  bI_EnableBalance                          : ARRAY[1..iCIk_NB_INKBALANCE] OF BOOL;    (*enable balance*)
  sI_InkDensitySet                          : ARRAY[1..iCIk_NB_INKBALANCE] OF REAL;    (*Ink density TO convert [kg] TO [liter]*)
  sI_CorrectionValue                        : ARRAY[1..iCIk_NB_INKBALANCE] OF REAL;    (*Correction value for the MUX retrieved data*)
  sI_WarningLevelSet                        : ARRAY[1..iCIk_NB_INKBALANCE] OF REAL;    (*warning level on the balance in [liter]*)
  sI_ErrorlevelSet                          : ARRAY[1..iCIk_NB_INKBALANCE] OF REAL;    (*error level on the balance in [liter]*)

  lR_VarParamScannerId                      : ARRAY[1..iCIk_NB_INKBALANCE] OF UDINT;   (*varnish parameter scanner ID*)
  iR_VarParamIndex                          : ARRAY[1..iCIk_NB_INKBALANCE] OF UINT;    (*varnish parameter index*)
  bR_VarParamCompatibility                  : ARRAY[1..iCIk_NB_INKBALANCE, 1..10] OF BOOL; (*varnish parameter compatibility to other index*)
  fR_VarParamTemp                           : ARRAY[1..iCIk_NB_INKBALANCE] OF REAL;    (*varnish parameter temperature*)
  fR_VarParamMenc                           : ARRAY[1..iCIk_NB_INKBALANCE] OF REAL;    (*varnish parameter meniscus*)
  aR_VarParamWaveform                       : ARRAY[1..iCIk_NB_INKBALANCE] OF STRING;  (*varnish parameter waveform*)
  iR_VarParamTimer                          : ARRAY[1..iCIk_NB_INKBALANCE] OF UINT;    (*varnish parameter timer*)
  fR_VarParamDensity                        : ARRAY[1..iCIk_NB_INKBALANCE] OF REAL;    (*varnish parameter density*)
  fR_VarParamViscosity                      : ARRAY[1..iCIk_NB_INKBALANCE] OF REAL;    (*varnish parameter viscosity*)
  iR_VarParamColorId                        : ARRAY[1..iCIk_NB_INKBALANCE] OF UINT;    (*varnish parameter color ID*)

  aI_CalibrateFrameText1                    : ARRAY[1..iCIk_NB_INKBALANCE] OF STRING;  (*Calibration string variable for text 1*)
  aI_CalibrateFrameText2                    : ARRAY[1..iCIk_NB_INKBALANCE] OF STRING;  (*Calibration string variable for text 2*)

  fR_BalanceOffset                          : ARRAY[1..iCIk_NB_INKBALANCE] OF REAL;   (*Calibration value for empty tank*)


(*Last entry----retain (remanent) variables of PRG_INK and realated modules*)
  aL_Pattern                                : UDINT;  (*check pattern for rem validity*)
END_STRUCT
END_TYPE

// ---- DUTs/Projects/Structures/ST_REM_VAR_M.TcDUT
TYPE ST_REM_VAR_M :
(*************************************************************************************************)
(*  FILENAME:    ST_REM_VAR_M.EXP                                                                *)
(*  PROJECT:     CALMAR PUPLC                                                                    *)
(*  COPYRIGHT:   All rights reserved (c) Wifag//Polytype, Fribourg/Switzerland (2016)            *)
(*  ENVIRONMENT: TwinCAT PLC                                                                     *)
(*  VERSION:     <version>                                                                       *)
(*************************************************************************************************)
(*  DESCRIPTION:                                                                   <description> *)
(*    Structure of remanent variables.                                                           *)
(*                                                                                </description> *)
(*************************************************************************************************)

STRUCT
  (*Clean Head*)
  (*************************************************************************************************)
  fRCH_Position_A                           : REAL;
  fRCH_Position_B                           : REAL;
  fRCH_Position_p1                          : REAL;
  fRCH_Position_p2                          : REAL;
  fRCH_PlaceSpeed                           : REAL;
  fRCH_WorkSpeed                            : REAL;
  fRCH_ServiceSpeed                         : REAL;

  lRCH_OffsetEncoder                        : DINT;
  

  lR_ToleranceLenPx                         : DINT;

(*Last entry----retain (remanent) variables of PRG_MACHINE and realated modules*)
  aL_Pattern                                : UDINT;  (*check pattern for rem validity*)
END_STRUCT
END_TYPE

// ---- DUTs/Projects/Structures/ST_REM_VAR_P.TcDUT
TYPE ST_REM_VAR_P :
(*************************************************************************************************)
(*  FILENAME:    ST_REM_VAR_P.EXP                                                                *)
(*  PROJECT:     CALMAR PUPLC                                                                    *)
(*  COPYRIGHT:   All rights reserved (c) Wifag//Polytype, Fribourg/Switzerland (2016)            *)
(*  ENVIRONMENT: TwinCAT PLC                                                                     *)
(*  VERSION:     <version>                                                                       *)
(*************************************************************************************************)
(*  DESCRIPTION:                                                                   <description> *)
(*    Structure of remanent variables.                                                           *)
(*                                                                                </description> *)
(*************************************************************************************************)

STRUCT
  (*PU*)
  //iL_ResolutionPhPx                      : ARRAY [1..iCPr_NB_PU] OF INT;    (*printhead pixel resolution [dpi]*)
  //fL_ResolutionEncoder                   : ARRAY [1..iCPr_NB_PU] OF LREAL;  (*resolution of encoder [um/increment]*)
  //iL_ResolutionSubPx                     : ARRAY [1..iCPr_NB_PU] OF INT;    (*subpixel pulse resolution [pulse/px]*)
  //fL_Pg_xOffset                          : ARRAY [1..iCPr_NB_PG] OF LREAL;  (*static offset of print group from start detection [m]*)
  //fL_Pg_vStartShiftFactor                : ARRAY [1..iCPr_NB_PU] OF LREAL;  (*shift of virtual start signal value from detection towards print group [m]*)
  //fL_Pg_vStartShiftOffset                : ARRAY [1..iCPr_NB_PU] OF LREAL;  (*shift of virtual start signal value from detection towards print group [m]*)
  //fL_SubstrateLen                        : ARRAY [1..iCPr_NB_PU] OF REAL;   (*length of substrate [m]*)

  bL_sAdsPrintUnit_bI_Enable             : ARRAY [1..iCPr_NB_PU] OF BOOL;
  lL_sAdsPrintUnit_sI_ShiftJobX          : ARRAY [1..iCPr_NB_PU] OF DINT;   (*Job(Unit) shift X in Pixel*)
  lL_sAdsPrintUnit_sI_ShiftJobY          : ARRAY [1..iCPr_NB_PU] OF DINT;   (*Job(Unit) shift Y in Pixel*)

  (*PM*)
  //fL_ResolutionEncoderPM                 : ARRAY [1..iCPr_NB_PM] OF LREAL;  (*resolution of encoder [um/increment]*)

  (*PG*)
  rL_sAdsPrintGroup_bI_Enable            : ARRAY [1..iCPr_NB_PG] OF BOOL;
  rL_sAdsPrintGroup_iO_PositionX         : ARRAY [1..iCPr_NB_PG] OF DINT;
  rL_sAdsPrintGroup_iO_StartPositionX    : ARRAY [1..iCPr_NB_PG] OF DINT;

  (*PC*)
  rL_sAdsPrintController                 : ARRAY [1..iCPr_NB_PC] OF BOOL;
  rL_sAdsPrintControllerHeater           : ARRAY [1..iCPr_NB_PC] OF BOOL;   (*Enable heater*)
  rL_sAdsPrintControllerPrint            : ARRAY [1..iCPr_NB_PC] OF BOOL;   (*Enable print*)

  (*PH*)
  rL_sAdsPrintHead_bI_Enable             : ARRAY [1..iCPr_NB_PH] OF BOOL;
  rL_sAdsPrintHead_iO_PositionX          : ARRAY [1..iCPr_NB_PH] OF DINT;
  rL_sAdsPrintHead_iO_StartPositionX     : ARRAY [1..iCPr_NB_PH] OF DINT;
  rL_sAdsPrintHead_iO_StartPositionY     : ARRAY [1..iCPr_NB_PH] OF DINT;
  rL_sAdsPrintHead_aI_MaskFileName       : ARRAY [1..iCPr_NB_PH] OF STRING; (*File name of sticking mask file*)
  rL_sAdsPrintHead_aI_WaveFileName       : ARRAY [1..iCPr_NB_PH] OF STRING; (*File name of waveform configuration file*)
  rL_sAdsPrintHead_fI_VoltScale          : ARRAY [1..iCPr_NB_PH] OF REAL;   (*File name of waveform configuration file*)
  
  bL_WithMark                            : BOOL;  (*use mark detection*)
  fL_MarkLength                          : REAL;  (*mark length*)
  fL_MarkHeigth                          : REAL;  (*mark width*)
  //fL_HeadGap                             : REAL;

  //bL_SpeedCompensationEnable             : BOOL;
  //fL_SpeedCompensationFactor             : REAL;
  //fL_SpeedCompensationBase               : REAL;

  fR_DriftTimeShift                      : LREAL;
  
  //iL_MonitorTempPH                       : INT;  (*Monitor level of temperature*)

(*Last entry----retain (remanent) variables of PRG_PRINT and realated modules*)
  aL_Pattern                             : UDINT;  (*check pattern for rem validity*)
END_STRUCT
END_TYPE

// ---- POUs/Products/Print_Weu/E_PosDomain.TcTLEO
{attribute 'qualified_only'}
{attribute 'strict'}
TYPE E_PosDomain :
(
	default := 0,
  master_pos := 1,
//  cycle_pos := 2
  pos_px      := 2     // position in [px]
) UINT;
END_TYPE

// ---- POUs/Products/Print_Weu/Mark/ST_MarkDefinition.TcDUT
TYPE ST_MarkDefinition :
STRUCT
  nId : DINT;             // mark id (array index)
  fHeight : LREAL;        // [m] mark height (size Y)
  fTrLength : LREAL;      // [m] triangle lenght
  fSqLength : LREAL;      // [m] square length ( square + triangle lengh = sizeX)
  fPosX : LREAL;          // [m] position X offset from 0/0
  fPosY : LREAL;          // [m] position Y offset from 0/0
  bInvertedX : BOOL;      // flipped in X axis (prior bMarksInverted)
  //bInvertedY : BOOL;      // flipped in Y axis
  //state
  sState : ST_MarkState;  // mark detection state
  //view
  bShow : BOOL;
  nMove : DINT;
END_STRUCT 
END_TYPE

// ---- POUs/Products/Print_Weu/Mark/ST_MarkState.TcDUT
TYPE ST_MarkState :
STRUCT
  bSet        : BOOL;     // mark was set & valid (detected)
  bMissed     : BOOL;     // mark was missing (+internally generated)
  bInArea     : BOOL;     // mark withing ok area
  dx          : LREAL;    // x displacement [m]
  dy          : LREAL;    // y displacement [m]
  fLengthReal : LREAL;    // real detected mark length [m]
  nPosXReal   : DINT;     // detected position X absolute [SubPx]
END_STRUCT
END_TYPE

// ---- POUs/Products/Print_Weu/ST_MappingDefinition.TcDUT
(*
  Hardware mapping definition.
*)
TYPE ST_MappingDefinition :
STRUCT
  // absolute hw mapping
  nPhInst : UDINT := 1;      // ph hw instance selection
  nPcInst : UDINT := 1;      // pc hw instance selection
  // module internal mapping (relative to given nPm)
  nPm     : UDINT := 1;      // to pm x
  nPg     : UDINT := 1;      // to pg in pm x
  nPa     : UDINT := 1;      // to pa in pg
  nPs     : UDINT := 1;      // to ps in pa
  nPc     : UDINT := 1;      // to pc in pm
  nPcCh   : UDINT := 1;      // to pc channel of pc 1-4
END_STRUCT
END_TYPE

// ---- POUs/Products/Print_Weu/ST_ModuleMachineInterface_IN.TcDUT
TYPE ST_ModuleMachineInterface_IN :
STRUCT
  // Inputs (from machine)
  bEStop                  : BOOL;             // EStop active
  bSleep                  : BOOL;             // Sleep active
  bSafetyCoverOk          : BOOL;             // Safety cover OK
  bServiceDoorsOk         : BOOL;             // Safety Doors OK
  bExhaustVacuumWarning   : BOOL;             // Vacuum warning level reached
  bExhaustVacuumError     : BOOL;             // Vacuum error level reached
  bExhaustFUError         : BOOL;             // ??? (obsolete?)
  bDriftControlError      : BOOL;             // (obsolete) remove?
  bDriftControlMissMarks  : BOOL;             // (obsolete) remove?
  bSafetyOk               : BOOL;              // generic safty ok
  
  // new
  bUnitInPrintPosition    : BOOL;             // Print module in print position
  bEngaged                : BOOL;             // Print module engaged
  bPrintEnabled           : BOOL;             // Printing enabled
  
  // other
  fSubstrateThickness     : LREAL := 0.000_1; // Substrate thickness [m]
  fSubstrateLen           : LREAL;            // Substrate length [m]
  fWebStretchCalculated   : LREAL;            // Web strech factor converted
  fLateralRegister        : LREAL;            // Lateral regster [m]
  fModule2ToModule3       : LREAL;            // Distance between Module 2 and 3 [m]
  bTargetSpeedReached     : BOOL;             // Target speed reached
  fNeutralFibreFactor     : LREAL;            // Neutral fibre factor [%]

END_STRUCT
END_TYPE

// ---- POUs/Products/Print_Weu/ST_ModuleMachineInterface_OUT.TcDUT
TYPE ST_ModuleMachineInterface_OUT :
STRUCT
  // Outputs (to Machine)
  fSpeed                : LREAL;            // Current module speed [m/s]
  bMoving               : BOOL;             // substrate/module is moving
  nPrintMarkPosBits     : WORD;             // Print mark position (bit coded)
  fMaxSpeed             : LREAL;            // Max. possible print module speed [m/s]
  bSpeedExeeded         : BOOL;             // Module speed exeeded;
END_STRUCT
END_TYPE

// ---- VISUs/Projects/Print/ST_ButtonFrameSel_Def.TcDUT
TYPE ST_ButtonFrameSel_Def :
STRUCT
  sImgId       : STRING;           // image id (to show)
  nFrameIdx    : UINT;             // frame index [0..x], index to select on click
  pFrameSelect : POINTER TO UINT;  // pointer to frame selection variable (variable to write to change the selected frame)
  sVisuName    : T_MaxString;      // visualisation name
END_STRUCT
END_TYPE

// ---- GVLs/Configuration/CONFIGURATION.TcGVL
{attribute 'Tc2GvlVarNames'}
VAR_GLOBAL CONSTANT
(*************************************************************************************************)
(*  FILENAME:    CONFIGURATION.EXP                                                               *)
(*  PROJECT:     CALMAR PUPLC                                                                    *)
(*  COPYRIGHT:   All rights reserved (c) Wifag//Polytype, Fribourg/Switzerland (2016)            *)
(*  ENVIRONMENT: TwinCAT PLC                                                                     *)
(*  VERSION:     <version>                                                                       *)
(*************************************************************************************************)
(*  DESCRIPTION:                                                                   <description> *)
(*    Configuration data system.                                                                 *)
(*                                                                                </description> *)
(*************************************************************************************************)

(*************************************************************************************************)
(*Configuration System*)
(*************************************************************************************************)
  iCSYS_GEN_BLOCK_MAP_CONFIG        : UINT := 0;   (*Configuration FB_GEN_BLOCK_MAPPING*)
                                                   (*Bit0: use extended block id then UINT :=  1; (iC_CFG_BIT_EXT_ID) *)


(*************************************************************************************************)
(*Configuration InkSystem*)
(*************************************************************************************************)

(*ADS*)
(*************************************************************************************************)
  iCIk_NB_BLOCK_TYPES               : INT := 10;   (*Number of different ADS block types*)


(*GENERAL*)
(*************************************************************************************************)
  (*Number of print station*)
  iCIk_NB_PRINT_STA                 : INT := 1;    (*Number of print station*)


(*DEGASSING*)
(*************************************************************************************************)
  iCIk_NB_DGAS                      : INT := 1;    (*Number of dgas controller*)

  bCIk_INK_DEGASSING_EXISTING       : BOOL := TRUE;  (*Degassing of ink existing*)


(*MENISCUS*)
(*************************************************************************************************)
  (*Number of menc controller*)
  iCIk_NB_MENC                      : INT := 1;    (*Number of menc controller*)

  (*Mapping main meniscus*)
  iCIk_MAP_MAIN_MENC_PURGE          : ARRAY [1..iCIk_NB_MENC] OF INT := [1];  (*Mapping main menc to purge controller*)

  (*Number of sub menc controller*)
  iCIk_NB_SUB_MENC                  : INT := 2;    (*Number of sub menc controller*)

  (*Number of menc controller per station*)
  iCIk_NB_MENC_STA                  : INT := 3;    (*Number of menc controller per station (iCIk_NB_MENC + iCIk_NB_SUB_MENC)*)

  (*Mapping sub meniscus*)
  iCIk_MAP_SUB_MENC_MAIN_MENC       : ARRAY [1..iCIk_NB_SUB_MENC] OF INT := [1,1];  (*Mapping sub menc to main menc*)
  iCIk_MAP_SUB_MENC_PURGE           : ARRAY [1..iCIk_NB_SUB_MENC] OF INT := [1,2];  (*Mapping sub menc to purge controller*)
  iCIk_MAP_SUB_MENC_HTG             : ARRAY [1..iCIk_NB_SUB_MENC] OF INT := [1,2];  (*Mapping sub menc to headertank group*)


(*PURGE - GLOBAL*)
(*************************************************************************************************)
  iCIk_NB_PURGE_CONTR               : INT := 2;    (*Number of purge controller*)
  iCIk_NB_PURGE_GROUP               : INT := 4;    (*Number of purge groups*)

  (*Purge controller existing*)
  bCIk_PURGE_CONTR_EXIST            : ARRAY [1..iCIk_NB_PURGE_CONTR] OF BOOL := [TRUE,TRUE];

  (*Purge group existing*)
  bCIk_PURGE_GROUP_EXIST            : ARRAY [1..iCIk_NB_PURGE_GROUP] OF BOOL := [TRUE,TRUE,TRUE,TRUE];

  (*Mapping purge group*)
  cCIk_MAP_PURGE_GROUP_CONTR        : ARRAY [1..iCIk_NB_PURGE_GROUP] OF BYTE := [1,1,2,2];  (*Mapping purge group to purge controller*)
  cCIk_MAP_PURGE_GROUP_PURGE_STA    : ARRAY [1..iCIk_NB_PURGE_GROUP] OF BYTE := [1,2,1,2];  (*Mapping purge group to purge station*)

  (*Purge for White is working with a special sequence*)
  bCIk_PURGE_CONTR_SEQUENCE         : ARRAY [1..iCIk_NB_PURGE_CONTR] OF BOOL := [FALSE,FALSE];
  bCIk_MAP_PURGE_CONTR_SEQ_MENC_NEG : ARRAY [1..iCIk_NB_PURGE_CONTR] OF BYTE := [2,2];
  bCIk_MAP_PURGE_CONTR_SEQ_MENC_POS : ARRAY [1..iCIk_NB_PURGE_CONTR] OF BYTE := [3,3];

  bCIk_PURGE_SEQUENCE_MAIN_VALVE    : BOOL := TRUE;   (*Use main or sub valve for sequence*)
  bCIk_PURGE_CONTROLLER_SEQUENTIAL  : BOOL := FALSE;  (*Purge controller process sequential*)
  bCIk_PURGE_CYCLE_CLOSE_PH_VALVE   : BOOL := FALSE;  (*Close valve PHin and PHout between the cycles*)
  bCIk_PURGE_PRESSURE_LINE          : BOOL := TRUE;   (*Purge pressure is connected direct to a pressure line*)


(*INK*)
(*************************************************************************************************)
  iCIk_NB_HEADERTANK                : INT := 4;       (*Number of headertanks*)
  iCIk_NB_HEADERTANK_GROUP          : INT := 2;       (*Number of headertank groups*)

  (*Headertank existing*)
  (*'White Recirculation','White front','White back','Cyan','Magenta','Yellow','Black'*)
  bCIk_HEADERTANK_EXIST             : ARRAY [1..iCIk_NB_HEADERTANK] OF BOOL := [ TRUE, TRUE, TRUE, TRUE];
  bCIk_HEADERTANK_FILL_CLEANER      : ARRAY [1..iCIk_NB_HEADERTANK] OF BOOL := [FALSE,FALSE,FALSE,FALSE];
  bCIk_HEADERTANK_REFUSE            : ARRAY [1..iCIk_NB_HEADERTANK] OF BOOL := [FALSE,FALSE,FALSE,FALSE];
  bCIk_HEADERTANK_CHANGE            : ARRAY [1..iCIk_NB_HEADERTANK] OF BOOL := [ TRUE, TRUE, TRUE, TRUE];
  bCIk_HEADERTANK_FILL              : ARRAY [1..iCIk_NB_HEADERTANK] OF BOOL := [ TRUE, TRUE, TRUE, TRUE];
  bCIk_HEADERTANK_FLUSH             : ARRAY [1..iCIk_NB_HEADERTANK] OF BOOL := [ TRUE, TRUE, TRUE, TRUE];

  (*Mapping headertank*)
  iCIk_MAP_HEADERTANK_DGAS          : ARRAY [1..iCIk_NB_HEADERTANK] OF INT := [1,1,1,1];  (*Mapping headertank to degass*)
  iCIk_MAP_HEADERTANK_MENC_STA      : ARRAY [1..iCIk_NB_HEADERTANK] OF INT := [2,2,3,3];  (*Mapping headertank to menc station*)
  iCIk_MAP_HEADERTANK_INK           : ARRAY [1..iCIk_NB_HEADERTANK] OF INT := [1,1,2,2];  (*Mapping headertank to ink*)
  iCIk_MAP_HEADERTANK_INK_LEVEL     : ARRAY [1..iCIk_NB_HEADERTANK] OF INT := [1,2,3,4];  (*Mapping headertank to ink level sensor*)
  iCIk_MAP_HEADERTANK_INK_PUMP      : ARRAY [1..iCIk_NB_HEADERTANK] OF INT := [1,2,3,4];  (*Mapping headertank to ink pump*)
  iCIk_MAP_HEADERTANK_PURGE_CONTR   : ARRAY [1..iCIk_NB_HEADERTANK] OF INT := [1,1,2,2];  (*Mapping headertank to purge controller*)
  iCIk_MAP_HEADERTANK_PURGE_GROUP   : ARRAY [1..iCIk_NB_HEADERTANK] OF INT := [1,2,3,4];  (*Mapping headertank to purge group*)
  iCIk_MAP_HEADERTANK_PURGE_GROUPIDX: ARRAY [1..iCIk_NB_HEADERTANK] OF INT := [1,2,1,2];  (*Mapping headertank to purge group*)
  iCIk_MAP_HEADERTANK_STORAGE_PUMP  : ARRAY [1..iCIk_NB_HEADERTANK] OF INT := [1,2,3,4];  (*Mapping headertank to storagetank pump*)
  iCIk_MAP_HEADERTANK_CLEANER_PUMP  : ARRAY [1..iCIk_NB_HEADERTANK] OF INT := [1,1,2,2];  (*Mapping headertank to cleaner pump*)
  iCIk_MAP_HEADERTANK_RETURN_FLOW   : ARRAY [1..iCIk_NB_HEADERTANK] OF INT := [1,1,2,2];  (*Mapping headertank to return flow*)
  iCIk_MAP_HEADERTANK_TEMP_CONTR    : ARRAY [1..iCIk_NB_HEADERTANK] OF INT := [1,2,3,4];  (*Mapping headertank to Temp controller*)
  iCIk_MAP_HEADERTANK_HT_GROUP      : ARRAY [1..iCIk_NB_HEADERTANK] OF INT := [1,1,2,2];  (*Mapping headertank to headertank group*)

  (*Storagetank*)
  iCIk_NB_INK                       : INT  := 2;    (*Number of ink*)
  iCIk_NB_INKSTORAGE_TANK           : INT  := 3;    (*Number of storage tanks incl conservation tank*)
  iCIk_NB_INKSTORAGE_TANK_MAX       : INT  := CalmarCompInkSystem.GVL_InkDef.iCIk_NB_INKSTORAGE_TANK_MAX;    (*Max number of storage tanks*)
  iCIk_NB_INKSTORAGE_TANK_MIXER     : INT  := 2;    (*Number of storage tank mixer (not existing here)*)
  iCIk_NB_INKSTORAGE_TANK_PUMP      : INT  := 4;    (*e.g. iCIk_NB_HEADERTANK*)
  iCIk_STORAGE_TANK_PUMP_SETPOINT   : BOOL := FALSE; (*Pump speed controlled by a set point or fix*)
  iCIk_MAP_STORAGE_TANK_BALANCE     : ARRAY [1..iCIk_NB_INK] OF INT := [1,2];  (*Mapping storage tank to balances*)

  (*Ink storage tank existing, order see aC_STORAGETANK_NAME_DETAIL*)
  bCIk_INKSTORAGE_TANK_EXIST        : ARRAY [1..iCIk_NB_INKSTORAGE_TANK] OF BOOL := [TRUE,TRUE,TRUE];
  bCIk_INKSTORAGE_MIXER_EXIST       : ARRAY [1..iCIk_NB_INKSTORAGE_TANK] OF BOOL := [FALSE,FALSE,FALSE];
  iCIk_MAP_INKSTORAGE_MIXER         : ARRAY [1..iCIk_NB_INKSTORAGE_TANK] OF INT  := [    1,    2,    3];
  bCIk_MIXER_FEEDBACK_EXIST         : BOOL := FALSE;


  (*Number of ink pumps*)
  iCIk_NB_INK_PUMPS                 : INT := 10;  (*Number of ink pumps in total*)

  iCIk_NB_CLEANER_PUMPS             : INT := 2;   (*Number of cleaner pumps*)
  iCIk_CLEANER_PUMP_SETPOINT        : ARRAY [1..iCIk_NB_CLEANER_PUMPS]     OF BOOL := [FALSE,FALSE];  (*Pump speed controlled by a set point or fix*)

  iCIk_NB_RETURN_FLOW_UNITS         : INT  := 2;      (*Number of retrun flow units*)
  iCIk_RETURN_FLOW_PUMP_SETPOINT    : BOOL := FALSE;  (*Pump speed controlled by a set point or fix*)

  (*Number of ink level sensor*)
  iCIk_NB_INK_LEVEL_SENSOR          : INT := 6;   (*Number of ink level sensor*)
	iCIk_NB_INK_LEVEL_SENSOR_CIRCL    : INT := 1;   (*Number of ink level sensor for circulation*)


(*TEMP*)
(*************************************************************************************************)
  (*Number of heating*)
  iCIk_NB_TEMP_CONTR                : INT := 8;   (*Sum number of heating controllers*)
  iCIk_NB_TEMP_HYS                  : INT := 8;   (*Number of heating controller with hysteris*)

  (*Mapping temp*)
  iCIk_MAP_TEMP_INK                 : ARRAY [1..iCIk_NB_TEMP_CONTR] OF INT := [1,1,2,2,1,1,2,2];  (*Mapping temp to ink*)
  iCIk_MAP_TEMP_HT                  : ARRAY [1..iCIk_NB_TEMP_CONTR] OF INT := [1,2,3,4,1,2,3,4];  (*Mapping temp to ink*)
  iCIk_MAP_TEMP_PG                  : ARRAY [1..iCIk_NB_TEMP_CONTR] OF INT := [1,2,3,4,1,2,3,4];  (*Mapping temp to print group*)

  
(*BALANCE*)
(*************************************************************************************************)
  bCIk_BALANCE_EXISTING             : BOOL := TRUE;  (*Balance system existing*)

  cCIk_NB_BALANCE_CHANNELS          : BYTE:= 8;   (*Number of balance channels per MUX*)
  iCIk_NB_INKBALANCE                : INT := 2;   (*Number of used balance channels*)
  iCIk_NB_BALANCE_MUX               : INT := 1;   (*Number of balance MUX*)

  cCIk_BALANCE_MUX_ID               : ARRAY [1..iCIk_NB_BALANCE_MUX, 0..2] OF BYTE := [48,48,49]; (*Balance ASCII MUX ID 001*)

  (*Balance channel existing*)
  bCIk_INKBALANCE_EXIST             : ARRAY [1..iCIk_NB_INKBALANCE] OF BOOL := [TRUE, TRUE];

  (*Mapping balance*)
  cCIk_MAP_BALANCE_BALANCE_MUX      : ARRAY [1..iCIk_NB_INKBALANCE] OF BYTE := [1,1];        (*Mapping balance/storage tank to balance MUX*)
  cCIk_MAP_BALANCE_BALANCE_CHANNEL  : ARRAY [1..iCIk_NB_INKBALANCE] OF BYTE := [0,1];        (*Mapping balance/storage tank to balance channel*)

  iCIk_NB_COUNT_SEND_WARNING        : INT := 3;       (*Count of 'send data error' messages till warning*)
  iCIk_NB_COUNT_MOTION_WARNING      : INT := 10000;   (*Count of 'in motion' messages till warning*)
  iCIk_NB_COUNT_NC_WARNING          : INT := 5;       (*Count of 'not connected' messages till warning*)

  (*Messages*)
  iCIk_NB_BALANCE_MSG               : INT := 15;      (*Number of messages per balance*)


//BALANCE wiedre altes System!
  (*If no balance system existing iCIk_NB_INKBALANCE should nevertheless set to >0*)
	(*Number of balance (at least 1 for dummy)*)
  iCIk_BALANCE_POWER_SUPPLY         : INT  := 5;     (*Power supply of balances [V]*)
	fCIk_BALANCE_RATED_OUTPUT         : REAL := 3.0;   (*[mV/V]*)
	fCIk_BALANCE_RATED_CAPACITY       : REAL := 10.0;  (*[kg]*)
	fCIk_BALANCE_REFUSE_FULL          : REAL := 9.0;   (*[kg]*)
	fCIk_BALANCE_CLEANER_EMPTY        : REAL := 1.0;  (*[kg]*)

  
(*************************************************************************************************)
(*Configuration Machine                                                                          *)
(*************************************************************************************************)

(*ADS*)
(*************************************************************************************************)
  iCMa_NB_BLOCK_TYPES               : INT := 3;    (*Number of different ADS block types*)


(*GENERAL*)
(*************************************************************************************************)
  (*DEVICE COUNT*)
  iCMa_NB_Ax                        : INT := 3;      (*Number of axes*)
  iCMa_NB_Cp                        : INT := 2;      (*Number of cleaning process controllers*)
  iCMa_NB_Ca                        : INT := 8;      (*Number of clean axes: 4 per module*)
  iCMa_NB_Ma                        : INT := 1;      (*Number of machines*)

  (*Mapping GROUP*)
  iCPr_MAP_Cp_CuAxis                : ARRAY [1..iCMa_NB_Cp] OF INT := [1,5];    (*Mapping cleaning process to CU axis ADS*)
  iCPr_MAP_Cp_ChAxis                : ARRAY [1..iCMa_NB_Cp] OF INT := [2,6];    (*Mapping cleaning process to CH axis ADS*)
  iCPr_MAP_Cp_PuAxis                : ARRAY [1..iCMa_NB_Cp] OF INT := [3,7];    (*Mapping cleaning process to PU axis ADS*)
  iCPr_MAP_Cp_InkInterface          : ARRAY [1..iCMa_NB_Cp] OF INT := [4,8];    (*Mapping cleaning process to ink interface ADS*)

  (*Messages*)
  iCMa_NB_MSG                       : INT := 31;    (*Number of messages per machine*)

END_VAR

// ---- GVLs/Configuration/Configuration_Print.TcGVL
//{attribute 'qualified_only'}
{attribute 'Tc2GvlVarNames'}
VAR_GLOBAL CONSTANT
(*************************************************************************************************)
(*Configuration Print*)
(*************************************************************************************************)

(*ADS*)
(*************************************************************************************************)
iCPr_NB_BLOCK_TYPES               : INT := 6;    (*Number of different ADS block types*)

(*Print*)
nC_PrintResolution                : UDINT := 600;     (*Print resolutions native*)
nC_SubPixelResolution             : UDINT := 32;      (*SubPixel resolution, resolution extension of print resolution*)
nC_MemorySectionWidth             : UDINT := 16#800;  (*NIOS Memory section width/height*)
nC_MemorySectionDepth             : UDINT := 16#6000; (*NIOS Memory section depth/length*)
nC_YShiftOffset                   : UDINT := (nC_MemorySectionWidth - GVL_PrintDef.RIGEN5.iC_Ph_Width) / 2;  // [px] 384px for RICOH_GEN5



(*DEVICE COUNT*)
iCPr_NB_PH                        : INT := 24;  (*Number of printheads*)
iCPr_NB_PC                        : INT := 8;   (*Number of printhead controllers*)
iCPr_NB_PG                        : INT := 4;   (*Number of printhead groups*)
iCPr_NB_PM                        : INT := 2;   (*Number of print modules*)
iCPr_NB_PU                        : INT := 1;   (*Number of print units*)
iCPr_NB_SUBSTRATE_DEVICES         : INT := 1;   (*Number of substrate control devices*)
iCPr_NB_ASPECT                    : INT := 1;   (*Number of aspect definitions*)

iCPr_PH_MAPPING                   : ARRAY[1..iCPr_NB_PH] OF ST_MappingDefinition := 
[ 
  // PM 1 - NOTE: nPC global, nPcPc per pc, other values relative to PM
  (nPhInst := 1,  nPcInst := 1, nPm := 1, nPg := 1, nPa := 1, nPs := 1, nPc := 1, nPcCh := 1),    // 1
  (nPhInst := 2,  nPcInst := 1, nPm := 1, nPg := 1, nPa := 1, nPs := 1, nPc := 1, nPcCh := 2),    // 2
  (nPhInst := 3,  nPcInst := 1, nPm := 1, nPg := 1, nPa := 1, nPs := 1, nPc := 1, nPcCh := 3),    // 3
  (nPhInst := 4,  nPcInst := 2, nPm := 1, nPg := 1, nPa := 1, nPs := 1, nPc := 2, nPcCh := 1),    // 4
  (nPhInst := 5,  nPcInst := 2, nPm := 1, nPg := 1, nPa := 1, nPs := 1, nPc := 2, nPcCh := 2),    // 5
  (nPhInst := 6,  nPcInst := 2, nPm := 1, nPg := 1, nPa := 1, nPs := 1, nPc := 2, nPcCh := 3),    // 6
  (nPhInst := 7,  nPcInst := 3, nPm := 1, nPg := 2, nPa := 1, nPs := 1, nPc := 3, nPcCh := 1),    // 7
  (nPhInst := 8,  nPcInst := 3, nPm := 1, nPg := 2, nPa := 1, nPs := 1, nPc := 3, nPcCh := 2),    // 8
  (nPhInst := 9,  nPcInst := 3, nPm := 1, nPg := 2, nPa := 1, nPs := 1, nPc := 3, nPcCh := 3),    // 9
  (nPhInst := 10, nPcInst := 4, nPm := 1, nPg := 2, nPa := 1, nPs := 1, nPc := 4, nPcCh := 1),    // 10
  (nPhInst := 11, nPcInst := 4, nPm := 1, nPg := 2, nPa := 1, nPs := 1, nPc := 4, nPcCh := 2),    // 11
  (nPhInst := 12, nPcInst := 4, nPm := 1, nPg := 2, nPa := 1, nPs := 1, nPc := 4, nPcCh := 3),    // 12
  // PM 2 - NOTE: nPC global, nPcPc per pc, other values relative to PM
  (nPhInst := 13, nPcInst := 5, nPm := 2, nPg := 1, nPa := 1, nPs := 1, nPc := 1, nPcCh := 1),    // 13
  (nPhInst := 14, nPcInst := 5, nPm := 2, nPg := 1, nPa := 1, nPs := 1, nPc := 1, nPcCh := 2),    // 14
  (nPhInst := 15, nPcInst := 5, nPm := 2, nPg := 1, nPa := 1, nPs := 1, nPc := 1, nPcCh := 3),    // 15
  (nPhInst := 16, nPcInst := 6, nPm := 2, nPg := 1, nPa := 1, nPs := 1, nPc := 2, nPcCh := 1),    // 16
  (nPhInst := 17, nPcInst := 6, nPm := 2, nPg := 1, nPa := 1, nPs := 1, nPc := 2, nPcCh := 2),    // 17
  (nPhInst := 18, nPcInst := 6, nPm := 2, nPg := 1, nPa := 1, nPs := 1, nPc := 2, nPcCh := 3),    // 18
  (nPhInst := 19, nPcInst := 7, nPm := 2, nPg := 2, nPa := 1, nPs := 1, nPc := 3, nPcCh := 1),    // 19
  (nPhInst := 20, nPcInst := 7, nPm := 2, nPg := 2, nPa := 1, nPs := 1, nPc := 3, nPcCh := 2),    // 20
  (nPhInst := 21, nPcInst := 7, nPm := 2, nPg := 2, nPa := 1, nPs := 1, nPc := 3, nPcCh := 3),    // 21
  (nPhInst := 22, nPcInst := 8, nPm := 2, nPg := 2, nPa := 1, nPs := 1, nPc := 4, nPcCh := 1),    // 22
  (nPhInst := 23, nPcInst := 8, nPm := 2, nPg := 2, nPa := 1, nPs := 1, nPc := 4, nPcCh := 2),    // 23
  (nPhInst := 24, nPcInst := 8, nPm := 2, nPg := 2, nPa := 1, nPs := 1, nPc := 4, nPcCh := 3)     // 24
];


(*UNIT*)
iCPr_NB_PG_UNIT                   : INT := 4;   (*Number of groups in unit1*)

(*Mapping MODULE*)
iCPr_MAP_PM_PG                    : ARRAY [1..iCPr_NB_PM] OF INT := [1,3];    (*Mapping print module to first printhead group*)

(*GROUP*)
iCPr_NB_PC_GROUP_MAX              : INT := 2;   (*Maximal number of printead controller per group*)
iCPr_NB_PC_GROUP1                 : INT := 2;   (*Number of printhead controllers per group*)
iCPr_NB_PC_GROUP                  : ARRAY [1..iCPr_NB_PG] OF INT := [2,2,2,2];    (*Number of printhead controllers per group*)

(*Mapping GROUP*)
iCPr_MAP_PG_PU                    : ARRAY [1..iCPr_NB_PG] OF INT := [1,1,1,1];    (*Mapping printhead group to print unit*)
iCPr_MAP_PG_PM                    : ARRAY [1..iCPr_NB_PG] OF INT := [1,1,2,2];    (*Mapping printhead group to print module*)
iCPr_MAP_PG_HTG                   : ARRAY [1..iCPr_NB_PG] OF INT := [1,1,2,2];    (*Mapping printhead group to headertank group*)

(*CONTROLLER*)
iCPr_NB_PH_PC                     : ARRAY [1..iCPr_NB_PC] OF INT := [3,3,3,3,3,3,3,3];  (*Number or printhead per controller*)

(*CONTROLLER existing, order see aC_PC_NAME_DETAIL*)
bCPr_PC_EXIST                     : ARRAY [1..iCPr_NB_PC] OF BOOL := [TRUE,TRUE,TRUE,TRUE,TRUE,TRUE,TRUE,TRUE];

(*Mapping CONTROLLER*)
iCPr_MAP_PC_PG                    : ARRAY [1..iCPr_NB_PC] OF INT := [1,1,2,2,3,3,4,4];  (*Mapping printhead controller to printhead group*)
iCPr_MAP_PC_PH                    : ARRAY [1..iCPr_NB_PC, 1..iCPr_NB_PH_PER_CONTROLLER] OF INT
                                                := [ 1,  3,  5, -1,
                                                     2,  4,  6, -1,
                                                     7,  9, 11, -1,
                                                     8, 10, 12, -1,
                                                    13, 15, 17, -1,
                                                    14, 16, 18, -1,
                                                    19, 21, 23, -1,
                                                    20, 22, 24, -1];   (*Mapping printhead controller to printhead*)
                                                (*ARRAY  --------------------------------------*)
                                                (*|          PC  1  2  3  4  5  6  7  8 *)
                                                (*|              |  |  |  |  |  |  |  | *)
                                                (*|Channel 1 - [ 1, 2, 7, 8,13,14,19,20]*)
                                                (*|        2 - [ 3, 4, 9,10,15,16,21,22]*)
                                                (*|        3 - [ 5, 6,11,12,17,18,23,24]*)
                                                (*|        4 - [-1,-1,-1,-1,-1,-1,-1,-1]*)
                                                
(*PRINTHEAD*)
iCPr_NB_PH_PER_CONTROLLER         : INT := 4;   (*!!!Number of printhead channel per controller board, hw spec*)

(*PRINTHEAD existing, order see aC_PH_NAME_DETAIL*)
bCPr_PH_EXIST                     : ARRAY [1..iCPr_NB_PH] OF BOOL := [TRUE,TRUE,TRUE,TRUE,TRUE,TRUE,TRUE,TRUE,TRUE,TRUE,TRUE,TRUE,TRUE,TRUE,TRUE,TRUE,TRUE,TRUE,TRUE,TRUE,TRUE,TRUE,TRUE,TRUE];

(*Mapping PRINTHEAD*)
iCPr_MAP_PH_PC                    : ARRAY [1..iCPr_NB_PH] OF INT  := [1,2,1,2,1,2,3,4,3,4,3,4,5,6,5,6,5,6,7,8,7,8,7,8];  (*Mapping printhead to printhead controller*)
cCPr_MAP_PH_PC_Index              : ARRAY [1..iCPr_NB_PH] OF BYTE := [1,1,2,2,3,3,1,1,2,2,3,3,1,1,2,2,3,3,1,1,2,2,3,3];  (*Mapping printhead to printhead controller index*)
iCPr_MAP_PH_HT                    : ARRAY [1..iCPr_NB_PH] OF INT  := [1,1,1,1,1,1,2,2,2,2,2,2,3,3,3,3,3,3,4,4,4,4,4,4];  (*Mapping printhead to headertank*)
iCPr_MAP_PH_PM                    : ARRAY [1..iCPr_NB_PH] OF INT  := [1,1,1,1,1,1,1,1,1,1,1,1,2,2,2,2,2,2,2,2,2,2,2,2];  (*Mapping printhead to print module*)

END_VAR

// ---- GVLs/Configuration/Definitions.TcGVL
{attribute 'Tc2GvlVarNames'}
VAR_GLOBAL CONSTANT
(*************************************************************************************************)
(*  FILENAME:    DEFINTIONS.EXP                                                                  *)
(*  PROJECT:     CALMAR PUPLC                                                                    *)
(*  COPYRIGHT:   All rights reserved (c) Wifag//Polytype, Fribourg/Switzerland (2016)            *)
(*  ENVIRONMENT: TwinCAT PLC                                                                     *)
(*  VERSION:     <version>                                                                       *)
(*************************************************************************************************)
(*  DESCRIPTION:                                                                   <description> *)
(*    Global variable constant.                                                                  *)
(*                                                                                </description> *)
(*************************************************************************************************)

  aC_NAME_PROJECT               : STRING   := 'DPST-1026-WEU2';
  aC_NAME_PRODUCT               : STRING   := 'WEU';
  aC_VERSION_PRODUCT            : STRING   := '01.000.000';
  iC_VERSION_PRODUCT            : INT      := 010000;

  sC_AMSNETID_LOCALHOST         : STRING   := '';                   (* AMS_NET_ID of Localhost *)
  sC_AMSNETID_IO                : STRING   := '172.17.2.140.3.1'; //'172.21.10.11.2.1';   (* AMS_NET_ID of IO *)

  aC_WifagDataPath              : STRING[255] := 'C:\ProgramData\WifagPolytype\';     (*Path of Wifag ProgramData*)
  aC_PlcSubPath                 : STRING[255] := 'PrintUnitPlc\02_Plc\';              (*Sub path to 02_PLC*)
  aC_RecipeSubPath              : STRING[255] := 'Recipe\';                           (*Sub path to recipe*)

  aC_PlcConfigPath              : STRING   := 'C:\ProgramData\WifagPolytype\WEUPrintUnitPlc\';   (*Plc config / report data path*)
  aC_PlcFlashFileSubPath        : STRING   := '03_Flash\';     (*firmware file sub-directory*)
  aC_PlcWaveformFileSubPath     : STRING   := '04_Waveform\';  (*waveform file sub-directory*)
  aC_PlcMaskFileSubPath         : STRING   := '05_Mask\';      (*stiching mask file sub-directory*)
  aC_PlcMapFileSubPath          : STRING   := '06_Map\';       (*correction map file sub-directory*)
  aC_PlcRecipeSubPath           : STRING   := '02_Plc\Recipe\';(*recipe file sub-directory*)  
  aC_PlcBlockIdSubPath          : STRING   := '02_Plc\BlockId\';(*blockId file sub-directory*)
  aC_PlcAlarmDbSubPath          : STRING   := '02_Plc\AlarmDb\';(*alarm db file sub-directory*)
  
  aC_PlcProjectCfgPath          : T_MaxString := 'C:\ProgramData\WifagPolytype\WEUPrintUnitPlc\02_Plc\DPST-1026-WEU 2 Demo\WEU2\PlcProject\Configuration\';
  
  
  iG_PC_ADDRESS                 : ARRAY[1..32] OF UINT := [1050,
                                                           1051,
                                                           1052,
                                                           1053,
                                                           1054,
                                                           1055,
                                                           1056,
                                                           1057,
                                                           1058,
                                                           1059];

END_VAR

// ---- GVLs/Configuration/GVL_TestCfg.TcGVL
{attribute 'qualified_only'}
VAR_GLOBAL CONSTANT
  //do_LibTest : BOOL := TRUE;
  do_TestStartUp : BOOL := TRUE;
END_VAR

// ---- GVLs/Configuration/REMANENT.TcGVL
{attribute 'Tc2GvlVarNames'}
VAR_GLOBAL PERSISTENT
(*************************************************************************************************)
(*  FILENAME:     REMANENT.EXP		                                                               *)
(*  PROJECT:      CALMAR Ink System                                                              *)
(*  COPYRIGHT:    Wifag//Polytype Fribourg	 		                                                 *)
(*  ENVIRONMENT:  TwinCAT PLC / CoDeSys	                                                         *)
(*	VERSION:			1.0																																						 *)
(*  DESCRIPTION:  Remanent Variables													        							             *)
(*																																															 *)
(*  AUTHOR:       PAR                                                                            *)
(*************************************************************************************************)
(*  MODIFICATIONS:                                                                               *)
(*************************************************************************************************)
(*  Date      Author  Comments                                                                   *)
(*  04.12.13  PAR     Initial Version                                                            *)
(*************************************************************************************************)

  (*Remanente Variablen*)
  sR_RemVar_P         : ST_REM_VAR_P;
  sR_RemVar_I        	: ST_REM_VAR_I;
	sR_RemVar_M					: ST_REM_VAR_M;
END_VAR

// ---- POUs/Products/Print_Weu/GVL_WEU.TcGVL
{attribute 'qualified_only'}
VAR_GLOBAL CONSTANT
  nC_WorkerPrintPerPm : UDINT := 2;
  nC_MaxPcPerPm : UDINT := 10;
  nC_MaxPhPerPm : UDINT := 40;
END_VAR

// ---- Version/Global_Version.TcGVL
{attribute 'TcGenerated'}
{attribute 'no-analysis'}
{attribute 'linkalways'}
// This function has been automatically generated from the project information.
VAR_GLOBAL CONSTANT
	{attribute 'const_non_replaced'}
	stLibVersion_PUPLC : ST_LibVersion := (iMajor := 1, iMinor := 1, iBuild := 0, iRevision := 0, nFlags := 0, sVersion := '1.1.0');
END_VAR

// ---- POUs/Products/Print_Weu/I_HardwarePool.TcIO
INTERFACE I_HardwarePool

METHOD registerPc : BOOL
VAR_INPUT
  pNewPc : POINTER TO FB_PC;
  //pAdsConfig  : POINTER TO FB_ADS_Config;
END_VAR
END_METHOD

METHOD registerPh : BOOL
VAR_INPUT
    pNewPh       : POINTER TO FB_PH;
    //pAdsConfig   : POINTER TO FB_ADS_Config;
    //pConnectedCb : POINTER TO CalmarCompPrint.FB_PC;
    //iChannel     : INT;
END_VAR
END_METHOD

END_INTERFACE

// ---- POUs/Products/Print_Weu/I_ModuleMaster.TcIO
INTERFACE I_ModuleMaster

PROPERTY iHardwarePool : I_HardwarePool
GET
END_GET
END_PROPERTY

PROPERTY iMasterPrintPosition : I_PrintPosition
GET
END_GET
END_PROPERTY

PROPERTY iWorkerParams : I_WorkerParams
GET
END_GET
END_PROPERTY

(*
  Register for PU StatusClient
*)
METHOD registerPuStatusClient : BOOL
VAR_INPUT
  sClient       : I_PrintStatusClient;
END_VAR
END_METHOD

METHOD registerPuSubystem : BOOL
VAR_INPUT
  iSubSys      : I_PrintSubsystem;
END_VAR
END_METHOD

END_INTERFACE

// ---- POUs/Products/Print_Weu/I_ProdManager.TcIO
INTERFACE I_ProdManager

END_INTERFACE

// ---- POUs/Products/Print_Weu/Mark/I_MarkDefinition.TcIO
INTERFACE I_MarkDefinition

(*
  Get a mark definition.
  nIdx= 1.._nMarks = registered marks
  nIdx= 0 - selects last mark 
  nIdx=-1 - selects boarder mark
*)
METHOD getMark : POINTER TO ST_MarkDefinition
VAR_INPUT
  nIdx : DINT; // mark index: 1.._nMarks, 0 = last (endMark) 
END_VAR
END_METHOD

(*Number of registered marks*)
PROPERTY nMarks : UDINT
GET
END_GET
END_PROPERTY

(*Number of detected marks*)
PROPERTY nMarksDetected : UDINT
GET
END_GET
END_PROPERTY

(*
  Register a mark to camera (teach)
*)
METHOD RegisterMark : BOOL
VAR_INPUT
  sMark : ST_MarkDefinition;
END_VAR
END_METHOD

METHOD ResetDefinition
END_METHOD

(*
  Reset all registered marks
*)
METHOD ResetMarkStates
END_METHOD

END_INTERFACE

// ---- POUs/Projects/InkSystem/PRG_INK.TcPOU
PROGRAM PRG_INK
(*************************************************************************************************)
(*  FILENAME:    PRG_INK.EXP                                                                     *)
(*  PROJECT:     CALMAR PUPLC                                                                    *)
(*  COPYRIGHT:   All rights reserved (c) Wifag//Polytype, Fribourg/Switzerland (2016)            *)
(*  ENVIRONMENT: TwinCAT PLC                                                                     *)
(*  VERSION:     <version>                                                                       *)
(*************************************************************************************************)
(*  DESCRIPTION:                                                                   <description> *)
(*    Controls the ink supply of digital printheads.                                             *)
(*    Main functions: Degassing, main and sub meniscus control, purge, ink supply, temperature   *)
(*    control, storage tank and mixer.                                                           *)
(*                                                                                </description> *)
(*************************************************************************************************)

VAR_INPUT
(*GENERAL*)
(*************************************************************************************************)
(*Interface to PRG_PRINT - direct accessed data*)
  pAdsPg                                      : ARRAY[1..iCPr_NB_PG] OF POINTER TO ST_ADS_PG;
  bPrgPrintIf_Ok                              : BOOL := FALSE;

(*Monitoring of terminals*)
  bI_Temperature1WcState                AT%I* : BOOL;                                  (*EL3204 temperature WcState*)
  bI_InkLevel1WcState                   AT%I* : BOOL;                                  (*EL3052 ink level WcState*)
  bI_Pressure1WcState                   AT%I* : BOOL;                                  (*EM3712 pressure WcState*)
  bI_Pressure2WcState                   AT%I* : BOOL;                                  (*EM3712 pressure WcState*)
  bI_SubPressureWcState                 AT%I* : ARRAY [1..iCIk_NB_SUB_MENC] OF BOOL;   (*EM3701 sub menc pressure WcState*)


(*DEGASSING*)
(*************************************************************************************************)
(*Inputs from hardware*)

(*Inputs from visu*)
  bIDp_EnableMainDgasValve                    : BOOL;                                  (*Enable main dgas valve*)


(*MENISCUS*)
(*************************************************************************************************)
(*Inputs from hardware*)


(*SUB MENISCUS*)
(*************************************************************************************************)
(*Inputs from hardware*)


(*PURGE - GLOBAL*)
(*************************************************************************************************)


(*VACUUM PUMP*)
(*************************************************************************************************)


(*INK*)
(*************************************************************************************************)


(*VARNISH*)
(*************************************************************************************************)
(*Inputs from hardware*)
  (*fill varnish*)
  bIKn_TankInkLevelReached              AT%I* : ARRAY [1..iCIk_NB_HEADERTANK] OF BOOL; (*-BX53, BX57: HT front level reached*)

  bIKn_TankCleanerLevelEmpty            AT%I* : BOOL; (*Tank cleaner level empty reached*)
  bIKn_TankRefuseLevelFull              AT%I* : BOOL; (*Tank refuse level full reached*)

(*Inputs from visu*)
  (*fill varnish ramp*)
  IIDp_MinDigitRampe                          : DINT := 1638;
  IIDp_MaxDigitRampe                          : DINT := 16383;
  fIDp_MinVoltRampe                           : REAL := 0;
  fIDp_MaxVoltRampe                           : REAL := 5;
  IIDp_MinPercentRampe                        : DINT := 0;
  IIDp_MaxPercentRampe                        : DINT := 100;
  IIDp_TimeRampe                              : DINT := 10;

  (*fill varnish pump*)
  wIDp_PumpTimeOffDelayVarnish                : WORD;                                  (*The time the pump runs [s]*)
  wIDp_MinSpeedFillInkPumpVarnish             : WORD;                                  (*Min limit of speed for fill varnish pump in percent*)
  wIDp_MaxSpeedFillInkPumpVarnish             : WORD;                                  (*Max limit of speed for fill varnish pump in percent*)
  wIDP_AnalogMaxDigitVarnish                  : WORD;                                  (*Max limit of speed for fill varnish pump in digits*)
  wIDP_AnalogMinDigitVarnish                  : WORD;                                  (*Min limit of speed for fill varnish pump in digits*)

  (*cleaner*)
  bIDp_StopFillCleaner                        : ARRAY [1..iCIk_NB_HEADERTANK]   OF BOOL;


(*TEMP*)
(*************************************************************************************************)
(*Inputs from hardware*)


(*BALANCE*)
(*************************************************************************************************)
  bI_Balance_AckInit                    AT%I* : BOOL;                                  (*EL6021: Balance acknowledge init*)
  bI_Balance_AckSend                    AT%I* : BOOL;                                  (*EL6021: Balance acknowledge send*)
  bI_Balance_DataRec                    AT%I* : BOOL;                                  (*EL6021: Balance receive data*)
  iI_Balance_RecDataLength              AT%I* : USINT;                                 (*EL6021: Balance receive data length*)
  cI_Balance_RxBuffWord                 AT%I* : ARRAY [0..49] OF UINT;                 (*EL6021: Data in 0..49*)
  bI_Balance_BufferFull                 AT%I* : BOOL;                                  (*EL6021: Balance buffer full*)
  bI_Balance_FramingError               AT%I* : BOOL;                                  (*EL6021: Balance framing error*)
  bI_Balance_OverRunError               AT%I* : BOOL;                                  (*EL6021: Balance over run error*)


(*BARCODE SCANNER*)
(*************************************************************************************************)
  bI_Barcode_AckInit                    AT%I* : BOOL;                                  (*EL6001: Barcode scanner acknowledge init*)
  bI_Barcode_AckSend                    AT%I* : BOOL;                                  (*EL6001: Barcode scanner acknowledge send*)
  bI_Barcode_DataRec                    AT%I* : BOOL;                                  (*EL6001: Barcode scanner receive data*)
  iI_Barcode_RecDataLength              AT%I* : USINT;                                 (*EL6001: Barcode scanner receive data length*)
  cI_Barcode_RxBuff                     AT%I* : ARRAY [0..21] OF BYTE;                 (*EL6001: Barcode scanner receive data buffer*)
  bI_Barcode_BufferFull                 AT%I* : BOOL;                                  (*EL6001: Barcode scanner buffer full*)
  bI_Barcode_FramingError               AT%I* : BOOL;                                  (*EL6001: Barcode scanner framing error*)
  bI_Barcode_OverRunError               AT%I* : BOOL;                                  (*EL6001: Barcode scanner over run error*)

  (*Simulation*)
  bSimulation                                 : BOOL;
END_VAR

VAR_OUTPUT
(*GENERAL*)
(*************************************************************************************************)
  bO_InitOk                                   : BOOL := FALSE;                         (*Init Ok*)
  bO_InkSystemOk                              : BOOL := TRUE;                          (*Global ink system status*)
  bO_InkStorageTankOk                         : BOOL := TRUE;                          (*Global ink storagetank status*)
  bO_TemperatureOk                            : BOOL;
  bO_VacuumOk                                 : BOOL;
  bO_StorageTankOk                            : BOOL;
  bO_TotalWcState                             : BOOL := FALSE;                         (*Monitoring: WcStates from all terminals*)
  bO_CommandPrintlineExec                     : ARRAY [1..iCIk_NB_HEADERTANK_GROUP] OF BOOL := [FALSE,FALSE];   (*Command printline is executing*)

  
(*DEGASSING*)
(*************************************************************************************************)
(*Outputs to hardware*)

(*Outputs to visu*)
  bODp_EnableMainDgasValve                    : BOOL;                                  (*enable main degass valve*)


(*MENISCUS*)
(*************************************************************************************************)
(*Outputs to hardware*)


(*SUB MENISCUS*)
(*************************************************************************************************)
(*Outputs to hardware*)


(*PURGE*)
(*************************************************************************************************)
  bO_MainPurgeReleaseValve   AT %Q* : BOOL;                        (*Main purge pressure release valve*)


(*VACUUM PUMP*)
(*************************************************************************************************)


(*INK*)
(*************************************************************************************************)
(*Outputs to hardware*)
  (*fill varnish*)
  bOKp_EnableFillInkPumpVarnish         AT%Q* : ARRAY [1..iCIk_NB_HEADERTANK] OF BOOL; (*Enable fill ink pump*)
  wOKp_StptSpeedFillInkPumpVarnish      AT%Q* : ARRAY [1..iCIk_NB_HEADERTANK] OF WORD; (*Setpoint of speed for fill ink pump*)

  bO_HTInkConnectionClose               AT%Q* : ARRAY [1..iCIk_NB_HEADERTANK] OF BOOL; (*-KX87: HT ink connection valve*)

  bO_RefuseValveHT                      AT%Q* : BOOL;  (*-KX63: White HT refuse valve*)                
  bO_RefuseValveStorageTank             AT%Q* : BOOL;  (*-KX67: White HT refuse to storage tank valve*)                

  bO_FlushingReturnPump                 AT%Q* : ARRAY [1..iCIk_NB_RETURN_FLOW_UNITS] OF BOOL;                

  (*Outputs to visu*)
  bODp_DgasPressOK                            : BOOL;  (*Dgas pressure ok*)

  (*White*)
  bO_WarnLevelEmptyRT                         : BOOL;  (*Empty level reached RT*)
  bO_ErrorLevelLowRT                          : BOOL;  (*Low level reached RT*)
  bO_ErrorLevelErrorRT                        : BOOL;  (*Error level reached RT*)
  bO_ErrorInkLossRT                           : BOOL;  (*Illogical ink loss RT*)
  bO_SupervisionFillPumpRT                    : BOOL;  (*Supervision fill pump RT*)
  bO_LevelRangePoint01RT                      : BOOL;  (*Level range 01 reached RT*)
  bO_RisingLevelRT                            : BOOL;  (*Level of RT rising*)

  bO_TankCleanerLevelEmpty                    : BOOL := FALSE;     (*Tank cleaner level empty reached*)
  bO_TankRefuseLevelFull                      : BOOL := FALSE;     (*Tank refuse level full reached*)
  

(*INKSTORAGE_TANK*)
(*************************************************************************************************)


(*TEMP*)
(*************************************************************************************************)
(*Outputs to hardware*)


(*BALANCE*)
(*************************************************************************************************)
  bO_Balance_ReqInit                    AT%Q* : BOOL;                            (*EL6021: Ctrl: Init request*)
  bO_Balance_ReqSend                    AT%Q* : BOOL;                            (*EL6021: Ctrl: Transmit request*)
  bO_Balance_AckRec                     AT%Q* : BOOL;                            (*EL6021: Ctrl: Receive accepted*)
  iO_Balance_SendDataLength             AT%Q* : USINT;                           (*EL6021: Ctrl: Output length*)
  cO_Balance_TxBuffWord                 AT%Q* : ARRAY [0..49] OF UINT;           (*EL6021: Data out 0..49*)


(*BARCODE SCANNER*)
(*************************************************************************************************)
  bO_Barcode_ReqInit                    AT%Q* : BOOL;                                  (*EL6001: Barcode scanner request init*)
  bO_Barcode_ReqSend                    AT%Q* : BOOL;                                  (*EL6001: Barcode scanner request send*)
  bO_Barcode_AckRec                     AT%Q* : BOOL;                                  (*EL6001: Barcode scanner acknowledge receive*)
  iO_Barcode_SendDataLength             AT%Q* : USINT;                                 (*EL6001: Barcode scanner send data length*)
  cO_Barcode_TxBuff                     AT%Q* : ARRAY [0..21] OF BYTE;                 (*EL6001: Barcode scanner send buffer*)
END_VAR

VAR
(*GENERAL*)
(*************************************************************************************************)
  (*Initiation*)
  bL_RemVar_Init                              : BOOL;

  (*Dummy read unused inputs*)
  bL_DummyReadInput                           : BOOL;
  iL_DummyReadInput                           : INT;

  (*Infos from other tasks*)
  sL_SystemCmd                                : ST_SYSTEM_CMD;                         (*PRG_MACHINE*)
  bL_CleanPumpRequest                         : ARRAY[1..iCIk_NB_SUB_MENC] OF BOOL;    (*PRG_MACHINE*)
  bL_CleanAfterPurge                          : ARRAY[1..iCIk_NB_SUB_MENC] OF BOOL;    (*PRG_MACHINE*)
  bL_CleanAbort                               : ARRAY[1..iCIk_NB_SUB_MENC] OF BOOL;    (*PRG_MACHINE*)
  bL_Engaged                                  : ARRAY[1..iCPr_NB_PM]       OF BOOL;    (*PRG_MACHINE*)
  bPU1Printing                                : BOOL;                                  (*PRG_PRINT*)

  iMachineInk                                 : ARRAY[1..iCPr_NB_PM] OF I_MachineInk;                          (*Interface to Machine*)


  (*Counter*)
  cL_State                                    : BYTE := cL_INIT;                       (*state init*)
  nTemp                                       : UDINT;
  nConvError                                  : UDINT;
  iL_Sel_BlkType                              : INT  := 1;                             (*used for module information visualisation*)
  iL_Counter                                  : INT;                                   (*working counter*)
  iL_Counter2                                 : INT;                                   (*working counter*)
  iL_Counter3                                 : INT;                                   (*working counter*)
  iL_Offset                                   : INT;                                   (*use for generic offsets*)
  iL_CounterDgas                              : INT;                                   (*Counter for Dgas controller*)
  iL_CounterMenc                              : INT;                                   (*Counter for Menc controller*)
  iL_CounterSubMenc                           : INT;                                   (*Counter for sub menc controller*)
  iL_CounterMencSta                           : INT;                                   (*Counter for menc controller*)
  iL_CounterPurge                             : INT;                                   (*Counter for purge controller*)
  iL_CounterPurgeGroup                        : INT;                                   (*Counter for purge group*)
  iL_CounterValve                             : INT;                                   (*Counter for Purge controller*)

  sC_Config_I                                 : ST_CONFIG_I;

(*INK SYSTEM ADS STRUCTURES *)
(*************************************************************************************************)
  sC_Ads_Info                                 : ST_ADS_INFO;                           (*ADS INFO*)
  sMappingInfo                                : T_MapInfo;        // Block mapping configuration
  ISystemBase                                 : I_SystemBase;     // reference to system base
  pModuleDef                                  : POINTER TO FB_ModuleDef;    // Module definition in system
  iSystemCmd                                  : I_SystemCmd;                // System Command interface
  iSystemStatus                               : I_SystemStatus;             // System Status interface
  
  sAdsIkHeaderTank                            : ARRAY[1..iCIk_NB_HEADERTANK]      OF ST_ADS_IK_HEADERTANK;
  sAdsIkHeaderTankGroup                       : ARRAY[1..iCIk_NB_HEADERTANK_GROUP]OF ST_ADS_HeaderTankGroup;

  sAdsIkInkPump                               : ARRAY[1..iCIk_NB_INK_PUMPS]       OF ST_ADS_IK_INKPUMP;

  sAdsIkDgas                                  : ARRAY[1..iCIk_NB_DGAS]            OF ST_ADS_PRESSION;

  sAdsIkMenc                                  : ARRAY[1..iCIk_NB_MENC_STA]        OF ST_ADS_PRESSION;

  sAdsIkPurgeController                       : ARRAY[1..iCIk_NB_PURGE_CONTR]     OF ST_ADS_IK_PURGE_CONTROLLER;

  sAdsIkPurgeGroup                            : ARRAY[1..iCIk_NB_PURGE_GROUP]     OF ST_ADS_IK_PURGE_GROUP;

  sAdsIkInkStorageTank                        : ARRAY[1..iCIk_NB_INKSTORAGE_TANK] OF ST_ADS_IK_INKSTORAGE_TANK;

  sAdsIkHeater                                : ARRAY[1..iCIk_NB_TEMP_CONTR]      OF ST_ADS_IK_HEATER;

  sAdsIkDummy                                 : ARRAY[1..1]                       OF ST_ADS_DUMMY;


  sL_Pressures                                : ST_IK_PRESSURE;
  sL_PumpConditions                           : ST_IK_INKPUMP_COND;
  sL_VacuumConditions                         : ST_IK_VACUUM_COND;

  
(*DEGASSING*)
(*************************************************************************************************)
  fb_DgasMencContr                            : ARRAY[1..iCIk_NB_DGAS] OF FB_MencController;
  fb_DgasValvePlus                            : ARRAY[1..iCIk_NB_DGAS] OF FB_ValveControl;    (*not existent*)
  fb_DgasPumpMinus                            : ARRAY[1..iCIk_NB_DGAS] OF FB_PumpControl;     (*MUC-MX123*)
  fb_DgasMainValve                            : ARRAY[1..iCIk_NB_DGAS] OF FB_ValveControl;    (*MUC-KX65*)
  fb_TofDgasMainValve                         : TOF;                                          (*Off timer for main dgas valve*)
  fb_VisuDgasMencController                   : FB_MencControllerVisu;


(*MENISCUS*)
(*************************************************************************************************)
                                                                                                  (*   mainW, mainCMYK, subW neg, subW pos,     subC,     subM,     subY, subK*)
  fb_MeniscusMencContr                        : ARRAY[1..iCIk_NB_MENC_STA] OF FB_MencController;
  fb_MeniscusValvePlus                        : ARRAY[1..iCIk_NB_MENC_STA] OF FB_ValveControl;    (*     -  ,      -  , MUW-KX73, MUW-KX77, MUC-KX71, MUC-KX73, MUC-KX75, MUC-KX77*)
  fb_MeniscusValveMinus                       : ARRAY[1..iCIk_NB_MENC_STA] OF FB_ValveControl;    (*MUW-KX61, MUC-KX61, MUW-KX71, MUW-KX75, MUC-KX72, MUC-KX74, MUC-KX76, MUC-KX78*)
  bL_EnableMencFromHeadertank                 : ARRAY[1..iCIk_NB_MENC_STA] OF BOOL;
  
  fb_MeniscusPump                             : FB_PumpControl;
  fb_VisuMeniscusMencController               : FB_MencControllerVisu;

  fb_TofRtLevelDetectionPoint04               : TOF;
  fb_SubMencShutOffValve                      : ARRAY[1..iCIk_NB_SUB_MENC] OF FB_ValveControl;    (*KX81, KX83*)
  bL_DeactivateSubMenc                        : ARRAY[1..iCIk_NB_SUB_MENC] OF BOOL;
  bL_SubMencShutOffValveForceFalse            : ARRAY[1..iCIk_NB_SUB_MENC] OF BOOL;
  bL_SubMencShutOffValveForceTrue             : ARRAY[1..iCIk_NB_SUB_MENC] OF BOOL;
  RF_TrigCleaning                             : ARRAY[1..iCIk_NB_SUB_MENC] OF RF_TRIG;
  R_TrigEnable                                : ARRAY[1..iCIk_NB_SUB_MENC] OF R_TRIG;
  fL_SubMencAdjustWhilePurgeClean             : ARRAY[1..iCIk_NB_SUB_MENC] OF REAL;  (*[mbar]*)

  
(*PURGE*)
(*************************************************************************************************)
  fb_PurgeController                          : ARRAY[1..iCIk_NB_PURGE_CONTR] OF FB_PurgeControllerSequence;  (*MUW-KX63, MUC-KX63*)
  fb_PurgeGroup                               : ARRAY[1..iCIk_NB_PURGE_GROUP] OF FB_PurgeGroup;               (*MUW-KX85, MUC-KX81, MUC-KX83, MUC-KX85, MUC-KX87*)

  bL_PurgeBusy                                : BOOL;
  fb_TofPurgeBusy                             : ARRAY[1..iCIk_NB_PURGE_CONTR] OF TOF;
  fb_PurgeControllerDummy                     : FB_PurgeController;  (*used for MencController if Purge is not relevant*)

  bL_PurgeDeAirValveRequest                   : ARRAY[1..iCIk_NB_HEADERTANK] OF BOOL; (*Request for DeAir valve*)

  bL_PurgeOutflow1ValveHT                     : ARRAY[1..iCIk_NB_HEADERTANK] OF BOOL; (*Enable outflow1 valve headertank*)
  bL_PurgeOutflow2ValveHT                     : ARRAY[1..iCIk_NB_HEADERTANK] OF BOOL; (*Enable outflow2 valve headertank*)

  bL_PurgeContrRequestHT                      : ARRAY[1..iCIk_NB_PURGE_CONTR] OF BOOL;
  bL_PurgeGroupRequestHT                      : ARRAY[1..iCIk_NB_PURGE_GROUP] OF BOOL;
  bL_PurgeGroupRequestDeAirHT                 : ARRAY[1..iCIk_NB_PURGE_GROUP] OF BOOL;

  
(*INK*)
(*************************************************************************************************)
(*controller*)
  fb_Headertank                               : ARRAY[1..iCIk_NB_HEADERTANK] OF FB_HEADERTANK_UNIT;

  bL_ChangeActiveOtherHT                      : ARRAY[1..iCIk_NB_HEADERTANK] OF BOOL;
  iL_Sel_HeaderTank                           : INT := 1;                              (*Selection for visu*)
  bL_CleanCommandToMachine                    : ARRAY[1..iCPr_NB_PM] OF BOOL;
  bL_CleanEnable1ToMachine                    : BOOL;
  bL_CleanEnable2ToMachine                    : BOOL;
  bL_CappingCommandToMachine                  : BOOL;
  bL_HeadertankCanEx                          : BOOL;
  bL_HeadertankFillCanEx                      : BOOL;
  lL_TimeReturnFlow                           : UDINT;
  tL_TimeReturnFlow                           : TIME;
  tL_TimeReturnFlowHt                         : ARRAY [1..iCIk_NB_HEADERTANK] OF TIME;
  tL_TimeBlowOut                              : TIME;
  lL_TimeBlowOut                              : UDINT;
  tL_TimeEmptyCleaner                         : TIME;
  lL_TimeEmptyCleaner                         : UDINT;
  lL_TimeWarnExchange                         : UDINT;
  tL_TimeMaxFill                              : TIME;
  wL_TimeMaxFillHt                            : ARRAY [1..iCIk_NB_HEADERTANK] OF WORD;
  fL_StorageTankLevelLiter                    : REAL;
  bL_Compatibility                            : BOOL;
  iL_ActIndex                                 : UINT;
  iL_StoragetankAssignmentIndex               : ARRAY [1..iCIk_NB_HEADERTANK] OF DINT;
  iL_ActStoragetankAssignmentIndex            : ARRAY [1..iCIk_NB_HEADERTANK] OF DINT;
  fb_RTrigChangeStateHeadertank               : ARRAY [1..iCIk_NB_HEADERTANK] OF R_TRIG;
  fb_RTrigCommandChangeHeadertank             : ARRAY [1..iCIk_NB_HEADERTANK] OF R_TRIG;       
  bL_BalanceMaintenanceExec                   : ARRAY [1..iCIk_NB_HEADERTANK] OF BOOL;
  sL_CommandChangePrintline                   : ARRAY [1..iCIk_NB_HEADERTANK_GROUP] OF ST_COMMAND;   (*Command to change printline system*)
  bL_CommandChangePrintlineVisu               : ARRAY [1..iCIk_NB_HEADERTANK_GROUP] OF BOOL;         (*Command to change printline system from visu*)
  bL_CommandChangePrintlinesVisu              : BOOL;                                                (*Command to change printlines system from visu*)
  fb_RTrigCommandChangePrintline              : ARRAY [1..iCIk_NB_HEADERTANK_GROUP] OF R_TRIG;       
  fb_FTrigCommandChangePrintline              : ARRAY [1..iCIk_NB_HEADERTANK_GROUP] OF F_TRIG;       
  sL_CommandEmptyPrintline                    : ARRAY [1..iCIk_NB_HEADERTANK_GROUP] OF ST_COMMAND;   (*Command to empty printline system*)
  bL_CommandEmptyPrintlineVisu                : ARRAY [1..iCIk_NB_HEADERTANK_GROUP] OF BOOL;         (*Command to empty printline system from visu*)
  bL_CommandEmptyPrintlinesVisu               : BOOL;                                                (*Command to empty printlines system from visu*)
  fb_RTrigCommandEmptyPrintline               : ARRAY [1..iCIk_NB_HEADERTANK_GROUP] OF R_TRIG;
  fb_FTrigCommandEmptyPrintline               : ARRAY [1..iCIk_NB_HEADERTANK_GROUP] OF F_TRIG;
  fb_RTrigCommandEmptyHT                      : ARRAY [1..iCIk_NB_HEADERTANK] OF R_TRIG;
  fb_FTrigCommandEmptyHT                      : ARRAY [1..iCIk_NB_HEADERTANK] OF F_TRIG;
  fb_RTrigCommandCleanerHT                    : ARRAY [1..iCIk_NB_HEADERTANK] OF R_TRIG;
  fb_FTrigCommandCleanerHT                    : ARRAY [1..iCIk_NB_HEADERTANK] OF F_TRIG;
  eL_LowestActiveStateChange                  : ARRAY [1..iCIk_NB_HEADERTANK_GROUP] OF EN_STATE_CHANGE;    (*Info to synchronize the states of the headertanks*)
  eL_LowestActiveStateEmpty                   : ARRAY [1..iCIk_NB_HEADERTANK_GROUP] OF EN_STATE_EMPTY;     (*Info to synchronize the states of the headertanks*)
  eL_LowestActiveStateFill                    : ARRAY [1..iCIk_NB_HEADERTANK_GROUP] OF EN_STATE_FILL;      (*Info to synchronize the states of the headertanks*)
  eL_LowestActiveStateFlush                   : ARRAY [1..iCIk_NB_HEADERTANK_GROUP] OF EN_STATE_FLUSH;     (*Info to synchronize the states of the headertanks*)
  eL_LowestActiveStateCleaning                : ARRAY [1..iCIk_NB_HEADERTANK_GROUP] OF EN_STATE_CLEANING;  (*Info to synchronize the states of the headertanks*)

  (*Fill varnish controller*)
  fb_FillInkVarnish                           : ARRAY [1..iCIk_NB_HEADERTANK] OF FB_INK_SUPPLY_UNIT;
  fb_Ramp                                     : ARRAY [1..iCIk_NB_HEADERTANK] OF FB_SPEED_RAMP;

  sL_InkTable                                 : ARRAY [1..iCIk_NB_HEADERTANK] OF ST_INKDEFINITON;  (*needed for VISU*)

  bL_TankInkLevelReachedVarnish               : ARRAY [1..iCIk_NB_HEADERTANK] OF BOOL; (*Tank ink level reached*)
  bL_LowLevelReached                          : ARRAY [1..iCIk_NB_HEADERTANK] OF BOOL; (*Tank ink low level reached*)
  bL_DgasPressOK                              : BOOL;                                  (*Dgas pressure ok*)

  (*Circulation ink controller*)
  fb_CirculationInk                           : ARRAY [1..iCIk_NB_HEADERTANK] OF FB_InkCirculation;


(*CLEANER*)
(*************************************************************************************************)
  (*White*)
  fb_Cleaner                                  : ARRAY [1..iCIk_NB_CLEANER_PUMPS] OF FB_CLEANER_UNIT;
  bL_CleanerPumpRequest                       : ARRAY [1..iCIk_NB_CLEANER_PUMPS] OF BOOL;  (*Cleaner pump request*)
  bL_CleanerPumpConfirmation                  : ARRAY [1..iCIk_NB_HEADERTANK]    OF BOOL;  (*Cleaner pump confirmation HT*)

  wIDp_AnalogMinPercentCleaner                : WORD := 0;     (*Min value analog-output in percent*)
  wIDp_AnalogMaxPercentCleaner                : WORD := 100;   (*Max value analog-output in percent*)
  wL_StptSpeedCleanInkPumpPercent             : WORD;          (*Setpoint cleaner pump in %*)
  wL_StptSpeedCleanInkPumpDigit               : WORD;          (*Setpoint cleaner pump in digit*)
  fL_MFunction                                : REAL := 0;     (*m of function for analog-output*)


(*RETURN FLOW*)
(*************************************************************************************************)
  fb_ReturnFlow                               : ARRAY [1..iCIk_NB_RETURN_FLOW_UNITS] OF FB_RETURN_FLOW_UNIT;
  fb_ReturnFlowStorTank                       : ARRAY [1..iCIk_NB_RETURN_FLOW_UNITS] OF FB_ValveControl; (*-KX35 to KX38: return flow valve*)

  bL_ReturnFlowRequest                        : ARRAY [1..iCIk_NB_RETURN_FLOW_UNITS] OF BOOL;  (*Return flow request*)
  iL_NbReturnFlowRequest                      : ARRAY [1..iCIk_NB_RETURN_FLOW_UNITS] OF UINT;  (*Number of return flow request*)
  iL_NbReturnFlowAssignHT                     : ARRAY [1..iCIk_NB_RETURN_FLOW_UNITS] OF UINT;  (*Number of assigned HT*)
  fb_TimerReturnFlow                          : ARRAY [1..iCIk_NB_RETURN_FLOW_UNITS] OF FB_TIMER_DUTYCYCLE;
  bL_ReturnFlowRefuse                         : ARRAY [1..iCIk_NB_RETURN_FLOW_UNITS] OF BOOL;  (*Return flow to refuse container*)
  fb_TonReturnFlowValveDelay                  : ARRAY [1..iCIk_NB_RETURN_FLOW_UNITS] OF TON;   (*Reset valves with a delay because pump request is controlled with a PWM.*)

  bL_ReturnFlowConfirmation                   : ARRAY [1..iCIk_NB_HEADERTANK]        OF BOOL;  (*Return flow confirmation HT*)




(*TEMP*)
(*************************************************************************************************)
(*temp controller*)
  fb_TempControllerHys                        : ARRAY [1..iCIk_NB_TEMP_HYS] OF FB_TempContrHysteresis; (*temp controller hysteresis*)
  bL_TemperatureWcState                       : ARRAY [1..iCIk_NB_TEMP_HYS] OF BOOL;                   (*EL3204 temperature WcState*)
  fb_RTrigEnableHeater                        : ARRAY [1..iCIk_NB_TEMP_HYS] OF R_TRIG;
  fb_RTrigDisableHeater                       : ARRAY [1..iCIk_NB_TEMP_HYS] OF R_TRIG;
  

(*INKSTORAGE_TANK*)
(*************************************************************************************************)
  fb_Storagetank                              : ARRAY [1..iCIk_NB_INKSTORAGE_TANK] OF FB_STORAGETANK_UNIT;
  bL_FillPumpConfirmation                     : ARRAY [1..iCIk_NB_HEADERTANK] OF BOOL;  (*Fill pump confirmation HT*)

	iL_Sel_InkStorTank	                        : INT := 1;
	fb_RTrigEnableInkStorTank                   : ARRAY [1..iCIk_NB_INKSTORAGE_TANK] OF R_TRIG; 	(*Start of enable ink storage tank*)
	fb_FTrigEnableInkStorTank                   : ARRAY [1..iCIk_NB_INKSTORAGE_TANK] OF F_TRIG; 	(*End of enable ink storage tank*)
	bL_OneInkStorTankEnabled                    : ARRAY [1..iCIk_NB_INKSTORAGE_TANK] OF BOOL;     (*Indicates that one ink storage tank is enabled*)
	bL_SeveralInkStorTanksEnabled               : ARRAY [1..iCIk_NB_INKSTORAGE_TANK] OF BOOL;     (*Indicates that several ink storage tanks are enabled*)
	bL_CheckNbInkStorTankEnabled                : ARRAY [1..iCIk_NB_INKSTORAGE_TANK] OF BOOL;     (**)
	iL_SelectedInkStorTank                      : ARRAY [1..iCIk_NB_INKSTORAGE_TANK] OF INT;      (*Selector for ink storage tank*)
	iL_SelectedInkStorTankLevel                 : ARRAY [1..iCIk_NB_INKSTORAGE_TANK] OF DINT;     (*Selector for ink storage tank level*)
	fb_TpStorTankSetZero                        : ARRAY [1..iCIk_NB_INKSTORAGE_TANK] OF TP;       (*Time to set balance to zero*)
	bL_MessageWarning                           : ARRAY [1..iCIk_NB_INKSTORAGE_TANK] OF BOOL;     (**)
	bL_MessageError                             : ARRAY [1..iCIk_NB_INKSTORAGE_TANK] OF BOOL;     (**)

	(*Messages*)
  fb_MsgQueueStorage                          : ARRAY [1..iCIk_NB_INKSTORAGE_TANK] OF FB_MSG_QUEUE;
	fb_BalanceMsgHandler                        : ARRAY [1..iCIk_NB_INKSTORAGE_TANK] OF FB_MSG_HANDLER;
	sL_MsgConfigStorage                         : ARRAY [1..iCIk_NB_INKSTORAGE_TANK] OF ST_MSG_CONFIG;

  bL_HtAssignedToStorage                      : ARRAY [1..iCIk_NB_INKSTORAGE_TANK] OF BOOL;

  (*Barcode scanner*)
  bI_EnableBarcodeScanner                     : BOOL;
  fb_BarcodeStoragetank                       : FB_BARCODE_COMM;


(*BALANCE*)
(*************************************************************************************************)
  FB_Balance                                  : ARRAY [1..iCIk_NB_INKBALANCE] OF FB_BALANCE_MONITOR;
  FB_BalanceLink                              : FB_BALANCE_COMM_WORD;
  bI_EnableBalanceLink                        : BOOL;                                  (*enable balance link communication*)
  bL_AckFaultGUI                              : BOOL;
  bL_BalanceOk                                : BOOL;

  fI_CorrectionValue                          : REAL := 1.0;                           (*Correction value for the MUX retrieved Data*)
  iI_RefreshRate                              : INT  := 2000;                          (*Balance Channel refresh rate in [ms]*)
  iI_MaintenanceTimeout                       : DINT := 5000;                          (*Maintenance Timout in [ms]*)

  iL_SelectedBalance                          : INT  := 1;                             (*Selector for balance channel, PLC VISU*)

  fL_BalanceOffset                            : ARRAY [1..iCIk_NB_INKBALANCE] OF REAL;

  (*Messages*)
  fB_BalanceMsg                               : ARRAY [1..iCIk_NB_INKSTORAGE_TANK, 1..iCIk_NB_BALANCE_MSG] OF FB_MESSAGE;

(*MIXER (not existing here)*)
(*************************************************************************************************)
  bL_MixerFeedbackExist                       : BOOL := FALSE;
  fL_MixerOnTime                              : REAL := 5.0;                                              (*Mixer on time [min]*)
  fL_MixerWaitTime                            : REAL := 1.0;                                              (*Mixer wait time [min]*)
  bL_MixerEnable                              : ARRAY [1..iCIk_NB_INKSTORAGE_TANK_MIXER] OF BOOL;         (*Mixer enable*)
  wL_MixerOnTime                              : ARRAY [1..iCIk_NB_INKSTORAGE_TANK_MIXER] OF WORD;         (*Mixer on time [min]*)
  wL_MixerWaitTime                            : ARRAY [1..iCIk_NB_INKSTORAGE_TANK_MIXER] OF WORD;         (*Mixer wait time [min]*)
  fb_TpMixerOn                                : ARRAY [1..iCIk_NB_INKSTORAGE_TANK_MIXER] OF TP;           (*Mixer on*)
  fb_TpMixerWait                              : ARRAY [1..iCIk_NB_INKSTORAGE_TANK_MIXER] OF TP;           (*Mixer wait*)
  fb_TonMixerSupervision                      : ARRAY [1..iCIk_NB_INKSTORAGE_TANK_MIXER] OF TON;          (*Mixer supervision*)
  fb_RTrigMixerPulse                          : ARRAY [1..iCIk_NB_INKSTORAGE_TANK_MIXER] OF R_TRIG;       (*Trigger mixer pulse*)
  bL_MixerPulseIndicator                      : ARRAY [1..iCIk_NB_INKSTORAGE_TANK_MIXER] OF BOOL;         (*Mixer pulse indicator*)
  bL_MixerPulseError                          : ARRAY [1..iCIk_NB_INKSTORAGE_TANK_MIXER] OF BOOL;         (*Mixer pulse error*)
  bL_StorageTankMixerError                    : ARRAY [1..iCIk_NB_INKSTORAGE_TANK]       OF BOOL;         (*Storage tank mixer error*)
  bL_AckMixerPulseError                       : ARRAY [1..iCIk_NB_INKSTORAGE_TANK]       OF BOOL;         (*Ack mixer pulse error*)


(* ADS Mappping *)
(*************************************************************************************************)
  iL_I                                        : INT;                                   (*instance counter*)
  iL_I2                                       : INT;                                   (*second instance counter for double loops*)
  sL_pI                                       : POINTER TO ST_MAP_BLK;                 (*pointer to module mapping instance*)
  iL_Ctr                                      : INT;                                   (*counter value*)
  iL_ActElmt                                  : INT;                                   (*actual array element*)
  pL_Ctr                                      : POINTER TO INT;                        (*pointer to mapping array index*)
  aL_Name                                     : STRING;                                (*Block string creation*)
  iL_NumModules                               : INT;                                   (*number of different block types*)
  cL_Module                                   : BYTE;                                  (*this module number*)

  FB_GEN_BLOCK_MAPPING                        : FB_GEN_BLOCK_MAPPING;                  (*generation of block mappings in this module*)
  Fb_RegToAry                                 : FB_REG_TO_ARY;

  sL_MOD_MAP                                  : ARRAY [1..iCIk_NB_BLOCK_TYPES] OF ST_MAP_MODBLKARY;  (*array conataining all modules with their mapping informations*)
  sL_ModBlkAry                                : ST_MAP_MODBLKARY;

  sL_BLK_PURGE_CONTR                          : ARRAY [1..iCIk_NB_PURGE_CONTR]     OF ST_MAP_BLK;
  sL_BLK_PURGE_GROUP                          : ARRAY [1..iCIk_NB_PURGE_GROUP]     OF ST_MAP_BLK;
  sL_BLK_DGAS                                 : ARRAY [1..iCIk_NB_DGAS]            OF ST_MAP_BLK;
  sL_BLK_MENC                                 : ARRAY [1..iCIk_NB_MENC_STA]        OF ST_MAP_BLK;
  sL_BLK_INKSTORAGE_TANK                      : ARRAY [1..iCIk_NB_INKSTORAGE_TANK] OF ST_MAP_BLK;
  sL_BLK_HEADERTANK                           : ARRAY [1..iCIk_NB_HEADERTANK]      OF ST_MAP_BLK;
  sL_BLK_HEADERTANK_GROUP                     : ARRAY [1..iCIk_NB_HEADERTANK_GROUP]OF ST_MAP_BLK;
  sL_BLK_INKPUMP                              : ARRAY [1..iCIk_NB_INK_PUMPS]       OF ST_MAP_BLK;
  sL_BLK_HEATER                               : ARRAY [1..iCIk_NB_TEMP_CONTR]      OF ST_MAP_BLK;
 
 (* FB to store the generated block ID's *)
  bL_ExecuteBlockIdSave                      : BOOL;
  fb_BlkIdSave                               : FB_BLK_ID_SAVE;

(*Automatic flushing device print unit*)
  iL_SelHeaderTankFlushing                   : INT := 1;                        (*Selection for visu*)
  aI_FlushingSafePattern                     : STRING;                          (*Safe pattern*)
  fb_TonFlushingUnlock                       : TON;
  bL_FlushingUnlock                          : BOOL;
  bL_FlushingHtEmpty                         : BOOL;
  bL_FlushingStop                            : BOOL;
  bL_FlushingActivate                        : BOOL;
  bL_FlushingActive                          : BOOL;
  bL_FlushingActiveHt                        : ARRAY [1..iCIk_NB_HEADERTANK] OF BOOL;
  fb_FTrigFlushingActive                     : F_TRIG;
  iL_FlushingState                           : INT;
  aL_FlushingState                           : STRING;
  bL_FlushingReturnFlowRequest               : ARRAY [1..iCIk_NB_HEADERTANK] OF BOOL;
  fb_FlushingReturnFlowTimer                 : FB_OperatingCounter;
  lL_OpCounterReturnFlowSeconds              : UDINT;
  lL_OpCounterReturnFlowCycles               : UDINT;

  (*Recipe read/write*)
  pFbRecipeMngr                              : POINTER TO FB_RECIPE_READ_WRITE;
    
  (*visu*)
  aVisuInkSystemFrameIndex                   : INT := 1;

  (*Simulation variables*)
  bL_SimInputs                               : BOOL := FALSE;
END_VAR

VAR CONSTANT
(*GENERAL*)
(*************************************************************************************************)
  cL_INIT                                     : BYTE := 0;       (*Init-state 0*)
  cL_INIT_PRG                                 : BYTE := 1;       (*Init-state 1*)
  cL_INIT_OK                                  : BYTE := 2;       (*Init-state 2*)

  iC_FilterSupervisionArraySize               : INT  := 50;      (*Amount of stored values*)
  iC_FilterSupervisionAddInfoArraySize        : INT  :=  4;      (*Amount of additional info for HT*)
END_VAR

VAR PERSISTENT
  lR_MinSpeedFillInkPumpCleaner               : WORD := 10;    (*Min limit of speed for cleaner pump*)
  lR_MaxSpeedFillInkPumpCleaner               : WORD := 100;   (*Max limit of speed for cleaner pump*)
  lR_AnalogMinDigitCleaner                    : WORD := 0;     (*Min value analog-output in digit*)
  lR_AnalogMaxDigitCleaner                    : WORD := 16383; (*Max value analog-output in digit*)
  lR_StptSpeedCleanInkPumpCleanerPercent      : WORD := 20;    (*Cleaner pump set point*)

  lL_TimeRefuseFlow                           : UDINT:= 5;
  tL_TimeRefuseFlow                           : TIME;

  (*Sub menc adjustment*)
  fR_SubMencSetAdjustWhilePurgeClean          : ARRAY [1..iCIk_NB_SUB_MENC] OF REAL;  (*[mbar]*)
  fR_SubMencSetTolWdwBig                      : REAL := 0.5;     (*TolWdwBig for sub menc while Purge/Clean [mbar]*)

  (*Automatic flushing device print unit*)
  lL_TimeFlushingReturnFlow                   : UDINT;
END_VAR

(*GENERAL*)
(*************************************************************************************************)
(*First action init call*)
IF NOT bO_InitOk THEN
  Init();
ELSE (*Else when init Ok*)
  (*Check interface*)
  IF bPrgPrintIf_Ok = FALSE THEN
    FOR iL_Counter := 1 TO iCPr_NB_PG DO
      bPrgPrintIf_Ok := TRUE;
      IF pAdsPg[iL_Counter] = 0 THEN bPrgPrintIf_Ok := FALSE; END_IF    // check ADS_PG access
    END_FOR
    RETURN;
  END_IF

  (*Dummy read unused inputs*)

  
  (*handle remanent variables*)
  RemVar();

  (*Automatic flushing device print unit*)
  (*Remove call after commissioning.*)
  //{warning 'Remove call AutoFlushingDevice after commissioning!!!'}
  AutoFlushingDevice();
  (*AuxReturnPump activation*)
  bO_FlushingReturnPump[1] := bL_FlushingReturnFlowRequest[1] OR bL_FlushingReturnFlowRequest[2];
  bO_FlushingReturnPump[2] := bL_FlushingReturnFlowRequest[3] OR bL_FlushingReturnFlowRequest[4];

  (*Call visualisation control*)
  Visu();

  (*Call simulation*)
  IF bSimulation THEN Simulate(); END_IF

  (*Set monitor variables, will be set to false if a device is not ok*)
  bO_VacuumOk      := TRUE;
  bO_TemperatureOk := TRUE;

  bO_TankCleanerLevelEmpty := NOT bIKn_TankCleanerLevelEmpty;
  bO_TankRefuseLevelFull   := NOT bIKn_TankRefuseLevelFull;

  (*Temp*)
  bL_TemperatureWcState[1]    := bI_Temperature1WcState;

  (*Infos from other tasks*)
  (*Machine infos are communicated via iMachineInk*)
  sL_SystemCmd                := PRG_MACHINE.sO_SystemCmd;
  bPU1Printing                := PRG_PRINT.FB_PU[ePr_PU_UNIT_1].sO_UnitStatus.bPrinting;
  FOR iL_Counter := 1 TO iCIk_NB_SUB_MENC DO
    bL_CleanPumpRequest[iL_Counter] := PRG_MACHINE.bO_CleanPumpRequest[iL_Counter];
    bL_CleanAfterPurge [iL_Counter] := PRG_MACHINE.sADS_CleanProcess[iL_Counter].bI_CleanAfterPurge;
    bL_CleanAbort      [iL_Counter] := PRG_MACHINE.sADS_CleanProcess[iL_Counter].bI_Abort;
  END_FOR
  FOR iL_Counter := 1 TO iCPr_NB_PM DO
    bL_Engaged[iL_Counter] := PRG_MACHINE.bL_IO_Engaged[iL_Counter];
  END_FOR

  (*Printline command and status for Change and Empty*)
  FOR iL_Counter := 1 TO iCIk_NB_HEADERTANK_GROUP DO
    sL_CommandChangePrintline[iL_Counter].bI_Command := sAdsIkHeaderTankGroup[iL_Counter].sI_CommandChangeInk.bI_Command;
    sL_CommandEmptyPrintline [iL_Counter].bI_Command := sAdsIkHeaderTankGroup[iL_Counter].sI_CommandEmptyInk .bI_Command;

    sAdsIkHeaderTankGroup[iL_Counter].sI_CommandChangeInk.bO_CommandCanEx := sL_CommandChangePrintline[iL_Counter].bO_CommandCanEx;
    sAdsIkHeaderTankGroup[iL_Counter].sI_CommandChangeInk.bO_CommandExec  := sL_CommandChangePrintline[iL_Counter].bO_CommandExec;
    sAdsIkHeaderTankGroup[iL_Counter].sI_CommandEmptyInk .bO_CommandCanEx := sL_CommandEmptyPrintline [iL_Counter].bO_CommandCanEx;
    sAdsIkHeaderTankGroup[iL_Counter].sI_CommandEmptyInk .bO_CommandExec  := sL_CommandEmptyPrintline [iL_Counter].bO_CommandExec;
  END_FOR


(*VACUUM*)
(*************************************************************************************************)
  (*DEGASSING*)
  FOR iL_CounterDgas := 1 TO iCIk_NB_DGAS DO
    fb_DgasMencContr[iL_CounterDgas]();
    fb_DgasValvePlus[iL_CounterDgas]();
    fb_DgasPumpMinus[iL_CounterDgas]();
    fb_DgasMainValve[iL_CounterDgas]();
  END_FOR
  bODp_DgasPressOK := fb_DgasMencContr[1].pErrorCode = 0;
  
  (*Output for main DGAS valve*)
  (*Valve should be activated all the time, except while sleep
  fb_TofDgasMainValve(IN := bIDp_EnableMainDgasValve, PT := T#15S);
  IF fb_TofDgasMainValve.Q THEN
    fb_DgasMainValve[1].mEnable();

    bODp_EnableMainDgasValve := TRUE;
  ELSE
    fb_DgasMainValve[1].mDisable();

    bODp_EnableMainDgasValve := FALSE;
	END_IF
  *)

  (*MENISCUS*)
  FOR iL_CounterMenc := 1 TO iCIk_NB_MENC_STA DO
    fb_MeniscusMencContr [iL_CounterMenc]();
    fb_MeniscusValvePlus [iL_CounterMenc]();
    fb_MeniscusValveMinus[iL_CounterMenc]();
    
    bO_VacuumOk := bO_VacuumOk AND fb_MeniscusMencContr[iL_CounterMenc].fb_2PointContrVacuum.bO_PressOk;
  END_FOR

  (*MAIN MENISCUS*)
  (*With the valve for minus the meniscus pump must also activated.*)
  IF fb_MeniscusValveMinus[1].pActive THEN
    fb_MeniscusPump.mEnable();
  ELSE
    fb_MeniscusPump.mDisable();
  END_IF
  fb_MeniscusPump();

  (*SUB MENISCUS*)
  FOR iL_CounterSubMenc := 1 TO iCIk_NB_SUB_MENC DO
    (*With the start of the cleaning the special setpoints are activated.*)
    (*With the end of the cleaning the original setpoints are reactivated.*)
    RF_TrigCleaning[iL_CounterSubMenc](CLK := bL_CleanPumpRequest[iL_CounterSubMenc]);

    (*Sub menc adjustment:*)
    (*- While Purge and Cleaning.*)
    (*  With a start of the Purge, the setpoint adjustment and the lI_TolWdwBig are set.*)
    IF     bL_CleanAfterPurge[iL_CounterSubMenc]
       AND (   iMachineInk[iCIk_MAP_SUB_MENC_HTG[iL_CounterSubMenc]].pPurgeRequest
            OR RF_TrigCleaning[iL_CounterSubMenc].RT
           ) 
    THEN
      (*Set adjusment value*)
      fL_SubMencAdjustWhilePurgeClean[iL_CounterSubMenc] := fR_SubMencSetAdjustWhilePurgeClean[iL_CounterSubMenc];
      (*Set lI_TolWdwBig*)
      fb_MeniscusMencContr[iCIk_NB_MENC + iL_CounterSubMenc].mSetToleranceBig(IbSetToleranceBig := TRUE, IfSetToleranceBig := fR_SubMencSetTolWdwBig);
    END_IF
  
    IF     (sAdsIkMenc[iCIk_NB_MENC + iL_CounterSubMenc].sI_PressSet.fI_Val <> 0) 
       AND (fL_SubMencAdjustWhilePurgeClean[iL_CounterSubMenc]              <> 0)
    THEN
      fb_MeniscusMencContr[iCIk_NB_MENC + iL_CounterSubMenc].pPressSetFactor :=   (  fL_SubMencAdjustWhilePurgeClean[iL_CounterSubMenc]
                                                                                   + sAdsIkMenc[iCIk_NB_MENC + iL_CounterSubMenc].sI_PressSet.fI_Val) 
                                                                                / sAdsIkMenc[iCIk_NB_MENC + iL_CounterSubMenc].sI_PressSet.fI_Val;
    ELSE
      fb_MeniscusMencContr[iCIk_NB_MENC + iL_CounterSubMenc].pPressSetFactor := 1;
    END_IF

    (*Rising trigger of enable sub menc conroller*)
    R_TrigEnable[iL_CounterSubMenc](CLK := sAdsIkMenc[iCIk_NB_MENC + iL_CounterSubMenc].bI_Enable);
    (*Reset values*)
    IF    R_TrigEnable[iL_CounterSubMenc].Q  (*(precaution)*)
       OR RF_TrigCleaning[iL_CounterSubMenc].FT
       OR bL_CleanAbort[iL_CounterSubMenc]
    THEN 
      (*Reset adjusment value*)
      fL_SubMencAdjustWhilePurgeClean[iL_CounterSubMenc] := 0; 
      (*Reset lI_TolWdwBig*)
      fb_MeniscusMencContr[iCIk_NB_MENC + iL_CounterSubMenc].mSetToleranceBig(IbSetToleranceBig := FALSE, IfSetToleranceBig := fR_SubMencSetTolWdwBig);
    END_IF
  END_FOR
    
(*TEMP*)
(*************************************************************************************************)
  (*Headertank, base plate heater*)
  FOR iL_Counter := 1 TO iCIk_NB_TEMP_HYS DO
    fb_RTrigEnableHeater[iL_Counter](CLK := bL_TemperatureWcState[iL_Counter]);
    IF fb_RTrigEnableHeater[iL_Counter].Q THEN
      fb_TempControllerHys[iL_Counter].mDisable();
    END_IF
    fb_RTrigDisableHeater[iL_Counter](CLK := NOT bL_TemperatureWcState[iL_Counter]);
    IF fb_RTrigDisableHeater[iL_Counter].Q THEN
      fb_TempControllerHys[iL_Counter].mEnable();
    END_IF
  
    fb_TempControllerHys[iL_Counter]();

    IF fb_TempControllerHys[iL_Counter].pErrorCode <> 0 THEN
      bO_TemperatureOk := FALSE;
		END_IF
  END_FOR


(*PURGE*)
(*************************************************************************************************)
  FOR iL_Counter := 1 TO iCIk_NB_PURGE_GROUP DO
    fb_PurgeController[cCIk_MAP_PURGE_GROUP_CONTR[iL_Counter]].IbPurgeGroupRequestHT     [cCIk_MAP_PURGE_GROUP_PURGE_STA[iL_Counter]] := bL_PurgeGroupRequestHT     [iL_Counter];
    fb_PurgeController[cCIk_MAP_PURGE_GROUP_CONTR[iL_Counter]].IbPurgeGroupRequestDeAirHT[cCIk_MAP_PURGE_GROUP_PURGE_STA[iL_Counter]] := bL_PurgeGroupRequestDeAirHT[iL_Counter];

    sAdsIkPurgeGroup[iL_Counter].bI_EnableFlush := FALSE;  (*Flush not existing*)
  END_FOR

  bL_PurgeBusy := FALSE;
  FOR iL_Counter := 1 TO iCIk_NB_PURGE_CONTR DO
    fb_PurgeController[iL_Counter].IbPurgeContrRequestHT := bL_PurgeContrRequestHT[iL_Counter];
    fb_PurgeController[iL_Counter]();

    (* TOF because pPurgeBusy is reset for one cycle if Purge is switching to the next HT.*)
    fb_TofPurgeBusy[iL_Counter](IN := fb_PurgeController[iL_Counter].pPurgeBusy, PT := T#20ms);
    bL_PurgeBusy := bL_PurgeBusy OR fb_TofPurgeBusy[iL_Counter].Q;
    iMachineInk[iL_Counter].pPurgeBusy := fb_TofPurgeBusy[iL_Counter].Q;
  END_FOR
  bO_MainPurgeReleaseValve := fb_PurgeController[1].bO_MainPurgeReleaseValve OR fb_PurgeController[2].bO_MainPurgeReleaseValve;
  

(*INK VARNISH*)
(*************************************************************************************************)
  (*Hadertank*)
  (******************)
  (*Inits*)
  FOR iL_Counter := 1 TO iCIk_NB_MENC_STA DO
    bL_EnableMencFromHeadertank[iL_Counter] := FALSE;
  END_FOR
  FOR iL_Counter := 1 TO iCIk_NB_PURGE_CONTR DO
    bL_PurgeContrRequestHT[iL_Counter] := FALSE;
  END_FOR
  FOR iL_Counter := 1 TO iCIk_NB_HEADERTANK_GROUP DO
    eL_LowestActiveStateChange  [iL_Counter] := eChangeEnd;
    eL_LowestActiveStateEmpty   [iL_Counter] := eEmptyEnd;
    eL_LowestActiveStateFill    [iL_Counter] := eFillEnd;
    eL_LowestActiveStateFlush   [iL_Counter] := eFlushEnd;
    eL_LowestActiveStateCleaning[iL_Counter] := eCleaningEnd;
  END_FOR

  (*Command for printline*)
  FOR iL_Counter := 1 TO iCIk_NB_HEADERTANK_GROUP DO
    fb_RTrigCommandChangePrintline[iL_Counter](CLK :=    sL_CommandChangePrintline[iL_Counter].bI_Command 
                                                      OR bL_CommandChangePrintlineVisu[iL_Counter]
                                                      OR bL_CommandChangePrintlinesVisu);
    fb_FTrigCommandChangePrintline[iL_Counter](CLK :=    sL_CommandChangePrintline[iL_Counter].bI_Command
                                                      OR bL_CommandChangePrintlineVisu[iL_Counter]
                                                      OR bL_CommandChangePrintlinesVisu);
  
    fb_RTrigCommandEmptyPrintline [iL_Counter](CLK :=    sL_CommandEmptyPrintline[iL_Counter].bI_Command 
                                                      OR bL_CommandEmptyPrintlineVisu[iL_Counter]
                                                      OR bL_CommandEmptyPrintlinesVisu);
    fb_FTrigCommandEmptyPrintline [iL_Counter](CLK :=    sL_CommandEmptyPrintline[iL_Counter].bI_Command
                                                      OR bL_CommandEmptyPrintlineVisu[iL_Counter]
                                                      OR bL_CommandEmptyPrintlinesVisu);
  END_FOR

  FOR iL_Counter := 1 TO iCIk_NB_HEADERTANK DO
    (*Change varnish not allowed if a change in another headertank is active.*)
    bL_ChangeActiveOtherHT[iL_Counter] := FALSE;
    FOR iL_Counter2 := 1 TO iCIk_NB_HEADERTANK DO
      IF iL_Counter <> iL_Counter2 THEN
        IF     sAdsIkHeaderTank[iL_Counter2].sI_CommandChange.bO_CommandExec 
           AND (iCIk_MAP_HEADERTANK_HT_GROUP[iL_Counter] = iCIk_MAP_HEADERTANK_HT_GROUP[iL_Counter2])
        THEN
          bL_ChangeActiveOtherHT[iL_Counter] := TRUE;
        END_IF
      END_IF
    END_FOR
  
    fb_RTrigChangeStateHeadertank[iL_Counter](CLK :=     sAdsIkHeaderTank[iL_Counter].bI_EnableFillInk
                                                     AND sAdsIkHeaderTank[iL_Counter].cO_StatusFillInk.5);
    IF fb_RTrigChangeStateHeadertank[iL_Counter].Q THEN
      fb_Headertank[iL_Counter].StateHeadertank := eHeadertankFull;
    END_IF

    fb_RTrigCommandChangeHeadertank[iL_Counter](CLK := sAdsIkHeaderTank[iL_Counter].sI_CommandChange.bI_Command);

    (*Allocate command for printline to headertank*)
    IF     (   fb_RTrigCommandChangePrintline[iCIk_MAP_HEADERTANK_INK[iL_Counter]].Q
            OR fb_RTrigCommandChangeHeadertank[iL_Counter].Q)
       AND bCIk_HEADERTANK_EXIST[iL_Counter]
    THEN
      (*Special profile for empty with ColorId = 255*)
      IF sAdsIkInkStorageTank[iL_StoragetankAssignmentIndex[iL_Counter]].sI_InkParameter.iColorId = sC_Config_I.iC_ColorIdEmpty THEN
        sAdsIkHeaderTank[iL_Counter].sI_CommandChange.bI_Command := FALSE;
        sAdsIkHeaderTank[iL_Counter].sI_CommandEmpty.bI_Command  := TRUE;
        fb_Headertank   [iL_Counter].bI_ExecutePurgeManu         := TRUE;
      (*Special storage tank with conservation*)
      ELSIF FIND(sAdsIkInkStorageTank[iL_StoragetankAssignmentIndex[iL_Counter]].aO_Name, sC_Config_I.aC_STORAGETANK_CONSERVATION) > 0 THEN
        sAdsIkHeaderTank[iL_Counter].sI_CommandChange.bI_Command   := FALSE;
        sAdsIkHeaderTank[iL_Counter].sI_CommandEmpty.bI_Command    := TRUE;
        sAdsIkHeaderTank[iL_Counter].sI_ActivateCleaner.bI_Command := TRUE;
        fb_Headertank   [iL_Counter].bI_ExecutePurgeManu           := TRUE;
      ELSE
        sAdsIkHeaderTank[iL_Counter].sI_CommandChange.bI_Command := TRUE;
        fb_Headertank   [iL_Counter].bI_ExecutePurgeManu         := FALSE;
      END_IF
    END_IF
    IF fb_FTrigCommandChangePrintline[iCIk_MAP_HEADERTANK_INK[iL_Counter]].Q THEN
      sAdsIkHeaderTank[iL_Counter].sI_CommandEmpty.bI_Command  := FALSE;
      sAdsIkHeaderTank[iL_Counter].sI_CommandChange.bI_Command := FALSE;
    END_IF
  
    IF     fb_RTrigCommandEmptyPrintline[iCIk_MAP_HEADERTANK_INK[iL_Counter]].Q 
       AND bCIk_HEADERTANK_EXIST[iL_Counter]
    THEN
      sAdsIkHeaderTank[iL_Counter].sI_CommandEmpty.bI_Command := TRUE;
      fb_Headertank   [iL_Counter].bI_ExecutePurgeManu        := TRUE;
    END_IF
    IF fb_FTrigCommandEmptyPrintline[iCIk_MAP_HEADERTANK_INK[iL_Counter]].Q THEN
      sAdsIkHeaderTank[iL_Counter].sI_CommandEmpty.bI_Command := FALSE;
    END_IF
  
    IF     fb_RTrigCommandEmptyHT[iL_Counter].Q 
       AND bCIk_HEADERTANK_EXIST[iL_Counter]
    THEN
      sAdsIkHeaderTank[iL_Counter].sI_CommandEmpty.bI_Command := TRUE;
      fb_Headertank   [iL_Counter].bI_ExecutePurgeManu        := TRUE;
    END_IF
    IF fb_FTrigCommandEmptyHT[iL_Counter].Q THEN
      sAdsIkHeaderTank[iL_Counter].sI_CommandEmpty.bI_Command := FALSE;
    END_IF
  
    (*Check states of all headertanks*)
    IF     (fb_Headertank[iL_Counter].StateChange > eChangeIdle)
       AND (fb_Headertank[iL_Counter].StateChange < eL_LowestActiveStateChange[iCIk_MAP_HEADERTANK_HT_GROUP[iL_Counter]])
    THEN
      eL_LowestActiveStateChange[iCIk_MAP_HEADERTANK_HT_GROUP[iL_Counter]] := fb_Headertank[iL_Counter].StateChange;
    END_IF
    IF     (fb_Headertank[iL_Counter].StateEmpty > eEmptyIdle)
       AND (fb_Headertank[iL_Counter].StateEmpty < eL_LowestActiveStateEmpty[iCIk_MAP_HEADERTANK_HT_GROUP[iL_Counter]])
    THEN
      eL_LowestActiveStateEmpty[iCIk_MAP_HEADERTANK_HT_GROUP[iL_Counter]] := fb_Headertank[iL_Counter].StateEmpty;
    END_IF
    IF     (fb_Headertank[iL_Counter].StateFill > eFillIdle)
       AND (fb_Headertank[iL_Counter].StateFill < eL_LowestActiveStateFill[iCIk_MAP_HEADERTANK_HT_GROUP[iL_Counter]])
    THEN
      eL_LowestActiveStateFill[iCIk_MAP_HEADERTANK_HT_GROUP[iL_Counter]] := fb_Headertank[iL_Counter].StateFill;
    END_IF
    IF     (fb_Headertank[iL_Counter].StateFlush > eFlushIdle)
       AND (fb_Headertank[iL_Counter].StateFlush < eL_LowestActiveStateFlush[iCIk_MAP_HEADERTANK_HT_GROUP[iL_Counter]])
    THEN
      eL_LowestActiveStateFlush[iCIk_MAP_HEADERTANK_HT_GROUP[iL_Counter]] := fb_Headertank[iL_Counter].StateFlush;
    END_IF
    IF     (fb_Headertank[iL_Counter].StateCleaning > eCleaningIdle)
       AND (fb_Headertank[iL_Counter].StateCleaning < eL_LowestActiveStateCleaning[iCIk_MAP_HEADERTANK_HT_GROUP[iL_Counter]])
    THEN
      eL_LowestActiveStateCleaning[iCIk_MAP_HEADERTANK_HT_GROUP[iL_Counter]] := fb_Headertank[iL_Counter].StateCleaning;
    END_IF

